LIN {X 0.037,Y -390.880,Z 705.624,A 0.000,B 0.000,C 90.000,E1 148.329} C_DIS
LIN {X -0.098,Y -391.913,Z 705.612,A 0.000,B 0.000,C 90.000,E1 146.215} C_DIS
LIN {X 0.024,Y -394.278,Z 705.595,A 0.000,B 0.000,C 90.000,E1 143.004} C_DIS
LIN {X 0.010,Y -397.554,Z 705.577,A 0.000,B 0.000,C 90.000,E1 139.828} C_DIS
LIN {X -0.151,Y -400.624,Z 705.563,A 0.000,B 0.000,C 90.000,E1 137.391} C_DIS
LIN {X -0.043,Y -401.218,Z 705.561,A 0.000,B 0.000,C 90.000,E1 137.025} C_DIS
LIN {X 0.071,Y -403.273,Z 705.556,A 0.000,B 0.000,C 90.000,E1 136.134} C_DIS
LIN {X -0.018,Y -403.782,Z 705.555,A 0.000,B 0.000,C 90.000,E1 135.972} C_DIS
LIN {X 0.110,Y -405.250,Z 705.553,A 0.000,B 0.000,C 90.000,E1 135.567} C_DIS
LIN {X -0.029,Y -408.274,Z 705.550,A 0.000,B 0.000,C 90.000,E1 135.040} C_DIS
LIN {X -0.096,Y -412.512,Z 705.547,A 0.000,B 0.000,C 90.000,E1 134.514} C_DIS
LIN {X 0.208,Y -421.421,Z 705.542,A 0.000,B 0.000,C 90.000,E1 133.542} C_DIS
LIN {X -0.002,Y -435.121,Z 705.535,A 0.000,B 0.000,C 90.000,E1 132.285} C_DIS
LIN {X 0.155,Y -448.848,Z 705.528,A 0.000,B 0.000,C 90.000,E1 131.067} C_DIS
LIN {X 0.075,Y -459.384,Z 705.523,A 0.000,B 0.000,C 90.000,E1 130.172} C_DIS
LIN {X -0.134,Y -469.829,Z 705.518,A 0.000,B 0.000,C 90.000,E1 129.277} C_DIS
LIN {X 0.058,Y -477.114,Z 705.514,A 0.000,B 0.000,C 90.000,E1 128.588} C_DIS
LIN {X 0.072,Y -486.841,Z 705.509,A 0.000,B 0.000,C 90.000,E1 127.649} C_DIS
LIN {X 0.054,Y -494.993,Z 705.505,A 0.000,B 0.000,C 90.000,E1 126.824} C_DIS
LIN {X -0.059,Y -501.689,Z 705.501,A 0.000,B 0.000,C 90.000,E1 126.137} C_DIS
LIN {X 0.320,Y -506.811,Z 705.498,A 0.000,B 0.000,C 90.000,E1 125.518} C_DIS
LIN {X 0.021,Y -510.602,Z 705.495,A 0.000,B 0.000,C 90.000,E1 125.105} C_DIS
LIN {X -0.156,Y -515.288,Z 705.492,A 0.000,B 0.000,C 90.000,E1 124.532} C_DIS
LIN {X -0.052,Y -520.560,Z 705.488,A 0.000,B 0.000,C 90.000,E1 123.785} C_DIS
LIN {X -0.281,Y -523.579,Z 705.485,A 0.000,B 0.000,C 90.000,E1 123.372} C_DIS
LIN {X -0.096,Y -528.125,Z 705.481,A 0.000,B 0.000,C 90.000,E1 122.625} C_DIS
LIN {X 0.290,Y -531.521,Z 705.478,A 0.000,B 0.000,C 90.000,E1 122.005} C_DIS
LIN {X -0.160,Y -535.306,Z 705.474,A 0.000,B 0.000,C 90.000,E1 121.337} C_DIS
LIN {X 0.156,Y -538.794,Z 705.470,A 0.000,B 0.000,C 90.000,E1 120.590} C_DIS
LIN {X -0.053,Y -543.188,Z 705.465,A 0.000,B 0.000,C 90.000,E1 119.617} C_DIS
LIN {X -0.177,Y -545.069,Z 705.462,A 0.000,B 0.000,C 90.000,E1 119.205} C_DIS
LIN {X 0.052,Y -549.671,Z 705.456,A 0.000,B 0.000,C 90.000,E1 118.052} C_DIS
LIN {X 0.114,Y -553.949,Z 705.450,A 0.000,B 0.000,C 90.000,E1 116.924} C_DIS
LIN {X -0.274,Y -557.841,Z 705.443,A 0.000,B 0.000,C 90.000,E1 115.848} C_DIS
LIN {X 0.106,Y -560.454,Z 705.439,A 0.000,B 0.000,C 90.000,E1 114.975} C_DIS
LIN {X -0.301,Y -562.053,Z 705.436,A 0.000,B 0.000,C 90.000,E1 114.463} C_DIS
LIN {X -0.060,Y -564.908,Z 705.430,A 0.000,B 0.000,C 90.000,E1 113.334} C_DIS
LIN {X -0.116,Y -566.717,Z 705.425,A 0.000,B 0.000,C 90.000,E1 112.514} C_DIS
LIN {X -0.032,Y -568.729,Z 705.419,A 0.000,B 0.000,C 90.000,E1 111.408} C_DIS
LIN {X 0.084,Y -570.665,Z 705.413,A 0.000,B 0.000,C 90.000,E1 110.301} C_DIS
LIN {X -0.170,Y -573.851,Z 705.402,A 0.000,B 0.000,C 90.000,E1 108.417} C_DIS
LIN {X -0.347,Y -576.446,Z 705.393,A 0.000,B 0.000,C 90.000,E1 106.804} C_DIS
LIN {X 0.230,Y -578.049,Z 705.387,A 0.000,B 0.000,C 90.000,E1 105.662} C_DIS
LIN {X -0.232,Y -580.067,Z 705.380,A 0.000,B 0.000,C 90.000,E1 104.356} C_DIS
LIN {X -0.237,Y -582.029,Z 705.372,A 0.000,B 0.000,C 90.000,E1 103.008} C_DIS
LIN {X -0.290,Y -584.774,Z 705.362,A 0.000,B 0.000,C 90.000,E1 101.130} C_DIS
LIN {X -0.218,Y -586.749,Z 705.354,A 0.000,B 0.000,C 90.000,E1 99.782} C_DIS
LIN {X 0.270,Y -588.417,Z 705.347,A 0.000,B 0.000,C 90.000,E1 98.398} C_DIS
LIN {X -0.113,Y -590.377,Z 705.338,A 0.000,B 0.000,C 90.000,E1 96.834} C_DIS
LIN {X 0.052,Y -592.186,Z 705.329,A 0.000,B 0.000,C 90.000,E1 95.220} C_DIS
LIN {X -0.008,Y -593.656,Z 705.322,A 0.000,B 0.000,C 90.000,E1 93.898} C_DIS
LIN {X 0.293,Y -594.679,Z 705.316,A 0.000,B 0.000,C 90.000,E1 92.808} C_DIS
LIN {X 0.237,Y -595.838,Z 705.308,A 0.000,B 0.000,C 90.000,E1 91.489} C_DIS
LIN {X 0.186,Y -596.766,Z 705.301,A 0.000,B 0.000,C 90.000,E1 90.172} C_DIS
LIN {X -0.081,Y -597.292,Z 705.295,A 0.000,B 0.000,C 90.000,E1 89.141} C_DIS
LIN {X 0.142,Y -597.849,Z 705.286,A 0.000,B 0.000,C 90.000,E1 87.535} C_DIS
LIN {X 0.138,Y -598.168,Z 705.279,A 0.000,B 0.000,C 90.000,E1 86.216} C_DIS
LIN {X -0.192,Y -598.390,Z 705.270,A 0.000,B 0.000,C 90.000,E1 84.666} C_DIS
LIN {X 0.221,Y -598.369,Z 705.264,A 0.000,B 0.000,C 90.000,E1 83.571} C_DIS
LIN {X 0.026,Y -598.147,Z 705.256,A 0.000,B 0.000,C 90.000,E1 82.008} C_DIS
LIN {X -0.165,Y -597.774,Z 705.250,A 0.000,B 0.000,C 90.000,E1 80.971} C_DIS
LIN {X -0.274,Y -597.248,Z 705.244,A 0.000,B 0.000,C 90.000,E1 79.926} C_DIS
LIN {X 0.300,Y -596.197,Z 705.235,A 0.000,B 0.000,C 90.000,E1 78.285} C_DIS
LIN {X -0.005,Y -595.130,Z 705.228,A 0.000,B 0.000,C 90.000,E1 76.992} C_DIS
LIN {X -0.033,Y -594.149,Z 705.222,A 0.000,B 0.000,C 90.000,E1 75.936} C_DIS
LIN {X 0.069,Y -593.162,Z 705.216,A 0.000,B 0.000,C 90.000,E1 74.866} C_DIS
LIN {X -0.146,Y -591.785,Z 705.209,A 0.000,B 0.000,C 90.000,E1 73.559} C_DIS
LIN {X 0.030,Y -589.941,Z 705.200,A 0.000,B 0.000,C 90.000,E1 71.945} C_DIS
LIN {X 0.242,Y -588.599,Z 705.194,A 0.000,B 0.000,C 90.000,E1 70.859} C_DIS
LIN {X -0.252,Y -586.709,Z 705.186,A 0.000,B 0.000,C 90.000,E1 69.571} C_DIS
LIN {X 0.117,Y -585.109,Z 705.180,A 0.000,B 0.000,C 90.000,E1 68.465} C_DIS
LIN {X -0.078,Y -583.265,Z 705.174,A 0.000,B 0.000,C 90.000,E1 67.411} C_DIS
LIN {X -0.167,Y -581.732,Z 705.170,A 0.000,B 0.000,C 90.000,E1 66.613} C_DIS
LIN {X -0.178,Y -579.515,Z 705.164,A 0.000,B 0.000,C 90.000,E1 65.537} C_DIS
LIN {X -0.073,Y -577.612,Z 705.160,A 0.000,B 0.000,C 90.000,E1 64.717} C_DIS
LIN {X -0.140,Y -574.784,Z 705.154,A 0.000,B 0.000,C 90.000,E1 63.640} C_DIS
LIN {X 0.009,Y -571.694,Z 705.147,A 0.000,B 0.000,C 90.000,E1 62.538} C_DIS
LIN {X 0.115,Y -568.247,Z 705.141,A 0.000,B 0.000,C 90.000,E1 61.435} C_DIS
LIN {X -0.237,Y -566.465,Z 705.138,A 0.000,B 0.000,C 90.000,E1 60.923} C_DIS
LIN {X -0.021,Y -563.520,Z 705.134,A 0.000,B 0.000,C 90.000,E1 60.078} C_DIS
LIN {X -0.042,Y -560.328,Z 705.129,A 0.000,B 0.000,C 90.000,E1 59.253} C_DIS
LIN {X 0.207,Y -557.352,Z 705.125,A 0.000,B 0.000,C 90.000,E1 58.535} C_DIS
LIN {X -0.055,Y -554.041,Z 705.122,A 0.000,B 0.000,C 90.000,E1 57.867} C_DIS
LIN {X -0.051,Y -550.348,Z 705.118,A 0.000,B 0.000,C 90.000,E1 57.168} C_DIS
LIN {X 0.253,Y -545.320,Z 705.113,A 0.000,B 0.000,C 90.000,E1 56.294} C_DIS
LIN {X 0.155,Y -542.697,Z 705.111,A 0.000,B 0.000,C 90.000,E1 55.881} C_DIS
LIN {X 0.063,Y -537.718,Z 705.107,A 0.000,B 0.000,C 90.000,E1 55.182} C_DIS
LIN {X -0.074,Y -534.597,Z 705.104,A 0.000,B 0.000,C 90.000,E1 54.769} C_DIS
LIN {X -0.076,Y -529.880,Z 705.101,A 0.000,B 0.000,C 90.000,E1 54.196} C_DIS
LIN {X -0.045,Y -524.667,Z 705.098,A 0.000,B 0.000,C 90.000,E1 53.623} C_DIS
LIN {X -0.063,Y -520.475,Z 705.096,A 0.000,B 0.000,C 90.000,E1 53.210} C_DIS
LIN {X -0.293,Y -516.009,Z 705.093,A 0.000,B 0.000,C 90.000,E1 52.844} C_DIS
LIN {X 0.063,Y -509.957,Z 705.091,A 0.000,B 0.000,C 90.000,E1 52.316} C_DIS
LIN {X -0.087,Y -505.088,Z 705.089,A 0.000,B 0.000,C 90.000,E1 51.984} C_DIS
LIN {X 0.054,Y -498.624,Z 705.086,A 0.000,B 0.000,C 90.000,E1 51.537} C_DIS
LIN {X -0.018,Y -490.654,Z 705.084,A 0.000,B 0.000,C 90.000,E1 51.045} C_DIS
LIN {X -0.006,Y -473.974,Z 705.078,A 0.000,B 0.000,C 90.000,E1 50.070} C_DIS
LIN {X 0.267,Y -454.288,Z 705.072,A 0.000,B 0.000,C 90.000,E1 48.852} C_DIS
LIN {X 0.001,Y -431.613,Z 705.064,A 0.000,B 0.000,C 90.000,E1 47.433} C_DIS
LIN {X -0.119,Y -422.494,Z 705.060,A 0.000,B 0.000,C 90.000,E1 46.782} C_DIS
LIN {X -0.020,Y -422.180,Z 705.060,A 0.000,B 0.000,C 90.000,E1 46.743} C_DIS
LIN {X -0.043,Y -422.169,Z 705.060,A 0.000,B 0.000,C 90.000,E1 46.743} C_DIS
LIN {X 0.214,Y -418.724,Z 705.049,A 0.000,B 0.000,C 90.000,E1 44.838} C_DIS
LIN {X -0.192,Y -409.471,Z 705.026,A 0.000,B 0.000,C 90.000,E1 40.620} C_DIS
LIN {X -0.082,Y -409.331,Z 705.024,A 0.000,B 0.000,C 90.000,E1 40.253} C_DIS
LIN {X 0.119,Y -409.487,Z 705.010,A 0.000,B 0.000,C 90.000,E1 37.810} C_DIS
LIN {X -0.114,Y -410.476,Z 704.993,A 0.000,B 0.000,C 90.000,E1 34.739} C_DIS
LIN {X -0.195,Y -411.108,Z 704.985,A 0.000,B 0.000,C 90.000,E1 33.372} C_DIS
LIN {X 0.026,Y -412.489,Z 704.970,A 0.000,B 0.000,C 90.000,E1 30.590} C_DIS
LIN {X 0.021,Y -413.990,Z 704.955,A 0.000,B 0.000,C 90.000,E1 27.847} C_DIS
LIN {X -0.006,Y -416.018,Z 704.938,A 0.000,B 0.000,C 90.000,E1 24.771} C_DIS
LIN {X -0.025,Y -417.955,Z 704.924,A 0.000,B 0.000,C 90.000,E1 22.386} C_DIS
LIN {X 0.140,Y -419.568,Z 704.915,A 0.000,B 0.000,C 90.000,E1 20.663} C_DIS
LIN {X 0.007,Y -421.974,Z 704.902,A 0.000,B 0.000,C 90.000,E1 18.308} C_DIS
LIN {X -0.081,Y -423.524,Z 704.894,A 0.000,B 0.000,C 90.000,E1 16.968} C_DIS
LIN {X 0.053,Y -426.313,Z 704.881,A 0.000,B 0.000,C 90.000,E1 14.592} C_DIS
LIN {X -0.033,Y -428.873,Z 704.870,A 0.000,B 0.000,C 90.000,E1 12.591} C_DIS
LIN {X 0.161,Y -431.052,Z 704.861,A 0.000,B 0.000,C 90.000,E1 10.894} C_DIS
LIN {X 0.139,Y -434.153,Z 704.848,A 0.000,B 0.000,C 90.000,E1 8.568} C_DIS
LIN {X -0.061,Y -436.899,Z 704.837,A 0.000,B 0.000,C 90.000,E1 6.606} C_DIS
LIN {X -0.198,Y -439.673,Z 704.826,A 0.000,B 0.000,C 90.000,E1 4.645} C_DIS
LIN {X -0.168,Y -441.687,Z 704.818,A 0.000,B 0.000,C 90.000,E1 3.326} C_DIS
LIN {X 0.175,Y -444.903,Z 704.807,A 0.000,B 0.000,C 90.000,E1 1.318} C_DIS
LIN {X -0.131,Y -448.220,Z 704.797,A 0.000,B 0.000,C 90.000,E1 359.484} C_DIS
LIN {X 0.198,Y -451.315,Z 704.788,A 0.000,B 0.000,C 90.000,E1 357.822} C_DIS
LIN {X 0.053,Y -455.759,Z 704.776,A 0.000,B 0.000,C 90.000,E1 355.584} C_DIS
LIN {X 0.099,Y -460.321,Z 704.763,A 0.000,B 0.000,C 90.000,E1 353.337} C_DIS
LIN {X -0.184,Y -463.478,Z 704.754,A 0.000,B 0.000,C 90.000,E1 351.781} C_DIS
LIN {X -0.078,Y -465.958,Z 704.747,A 0.000,B 0.000,C 90.000,E1 350.500} C_DIS
LIN {X -0.111,Y -468.963,Z 704.738,A 0.000,B 0.000,C 90.000,E1 348.926} C_DIS
LIN {X 0.083,Y -471.257,Z 704.731,A 0.000,B 0.000,C 90.000,E1 347.645} C_DIS
LIN {X 0.181,Y -474.654,Z 704.721,A 0.000,B 0.000,C 90.000,E1 345.755} C_DIS
LIN {X 0.061,Y -477.553,Z 704.712,A 0.000,B 0.000,C 90.000,E1 344.212} C_DIS
LIN {X -0.015,Y -480.523,Z 704.704,A 0.000,B 0.000,C 90.000,E1 342.670} C_DIS
LIN {X 0.098,Y -484.927,Z 704.692,A 0.000,B 0.000,C 90.000,E1 340.496} C_DIS
LIN {X 0.056,Y -490.130,Z 704.678,A 0.000,B 0.000,C 90.000,E1 338.050} C_DIS
LIN {X 0.114,Y -491.805,Z 704.675,A 0.000,B 0.000,C 90.000,E1 337.433} C_DIS
LIN {X 0.130,Y -493.357,Z 704.672,A 0.000,B 0.000,C 90.000,E1 336.975} C_DIS
LIN {X 0.172,Y -494.686,Z 704.671,A 0.000,B 0.000,C 90.000,E1 336.666} C_DIS
LIN {X 0.218,Y -496.414,Z 704.669,A 0.000,B 0.000,C 90.000,E1 336.357} C_DIS
LIN {X -0.136,Y -500.322,Z 704.666,A 0.000,B 0.000,C 90.000,E1 335.921} C_DIS
LIN {X 0.058,Y -507.384,Z 704.663,A 0.000,B 0.000,C 90.000,E1 335.281} C_DIS
LIN {X -0.130,Y -514.500,Z 704.660,A 0.000,B 0.000,C 90.000,E1 334.793} C_DIS
LIN {X -0.057,Y -527.150,Z 704.655,A 0.000,B 0.000,C 90.000,E1 333.948} C_DIS
LIN {X 0.013,Y -537.986,Z 704.651,A 0.000,B 0.000,C 90.000,E1 333.204} C_DIS
LIN {X 0.154,Y -543.938,Z 704.649,A 0.000,B 0.000,C 90.000,E1 332.743} C_DIS
LIN {X 0.171,Y -549.794,Z 704.646,A 0.000,B 0.000,C 90.000,E1 332.281} C_DIS
LIN {X -0.049,Y -555.364,Z 704.643,A 0.000,B 0.000,C 90.000,E1 331.820} C_DIS
LIN {X 0.078,Y -559.491,Z 704.641,A 0.000,B 0.000,C 90.000,E1 331.435} C_DIS
LIN {X 0.122,Y -566.010,Z 704.638,A 0.000,B 0.000,C 90.000,E1 330.795} C_DIS
LIN {X 0.253,Y -572.386,Z 704.634,A 0.000,B 0.000,C 90.000,E1 330.127} C_DIS
LIN {X -0.018,Y -578.608,Z 704.631,A 0.000,B 0.000,C 90.000,E1 329.488} C_DIS
LIN {X 0.281,Y -585.780,Z 704.626,A 0.000,B 0.000,C 90.000,E1 328.663} C_DIS
LIN {X -0.239,Y -595.015,Z 704.620,A 0.000,B 0.000,C 90.000,E1 327.661} C_DIS
LIN {X 0.105,Y -601.689,Z 704.616,A 0.000,B 0.000,C 90.000,E1 326.834} C_DIS
LIN {X -0.133,Y -605.781,Z 704.613,A 0.000,B 0.000,C 90.000,E1 326.342} C_DIS
LIN {X -0.014,Y -611.762,Z 704.609,A 0.000,B 0.000,C 90.000,E1 325.548} C_DIS
LIN {X 0.032,Y -616.458,Z 704.605,A 0.000,B 0.000,C 90.000,E1 324.895} C_DIS
LIN {X 0.083,Y -622.649,Z 704.600,A 0.000,B 0.000,C 90.000,E1 323.989} C_DIS
LIN {X 0.216,Y -627.607,Z 704.596,A 0.000,B 0.000,C 90.000,E1 323.210} C_DIS
LIN {X -0.113,Y -632.970,Z 704.591,A 0.000,B 0.000,C 90.000,E1 322.351} C_DIS
LIN {X 0.003,Y -638.866,Z 704.585,A 0.000,B 0.000,C 90.000,E1 321.331} C_DIS
LIN {X -0.301,Y -644.423,Z 704.580,A 0.000,B 0.000,C 90.000,E1 320.356} C_DIS
LIN {X -0.039,Y -649.734,Z 704.574,A 0.000,B 0.000,C 90.000,E1 319.337} C_DIS
LIN {X 0.182,Y -655.946,Z 704.567,A 0.000,B 0.000,C 90.000,E1 318.081} C_DIS
LIN {X 0.082,Y -660.015,Z 704.563,A 0.000,B 0.000,C 90.000,E1 317.229} C_DIS
LIN {X 0.019,Y -663.227,Z 704.558,A 0.000,B 0.000,C 90.000,E1 316.500} C_DIS
LIN {X 0.000,Y -667.217,Z 704.553,A 0.000,B 0.000,C 90.000,E1 315.526} C_DIS
LIN {X 0.021,Y -671.839,Z 704.546,A 0.000,B 0.000,C 90.000,E1 314.312} C_DIS
LIN {X 0.115,Y -675.298,Z 704.541,A 0.000,B 0.000,C 90.000,E1 313.338} C_DIS
LIN {X -0.191,Y -679.496,Z 704.534,A 0.000,B 0.000,C 90.000,E1 312.162} C_DIS
LIN {X -0.035,Y -682.652,Z 704.529,A 0.000,B 0.000,C 90.000,E1 311.191} C_DIS
LIN {X -0.225,Y -685.529,Z 704.524,A 0.000,B 0.000,C 90.000,E1 310.253} C_DIS
LIN {X -0.125,Y -686.898,Z 704.521,A 0.000,B 0.000,C 90.000,E1 309.769} C_DIS
LIN {X -0.252,Y -689.277,Z 704.516,A 0.000,B 0.000,C 90.000,E1 308.830} C_DIS
LIN {X -0.030,Y -690.417,Z 704.513,A 0.000,B 0.000,C 90.000,E1 308.338} C_DIS
LIN {X -0.041,Y -692.780,Z 704.506,A 0.000,B 0.000,C 90.000,E1 307.156} C_DIS
LIN {X 0.119,Y -694.865,Z 704.500,A 0.000,B 0.000,C 90.000,E1 305.964} C_DIS
LIN {X 0.095,Y -696.266,Z 704.495,A 0.000,B 0.000,C 90.000,E1 305.025} C_DIS
LIN {X -0.083,Y -697.758,Z 704.488,A 0.000,B 0.000,C 90.000,E1 303.865} C_DIS
LIN {X -0.137,Y -698.550,Z 704.484,A 0.000,B 0.000,C 90.000,E1 303.166} C_DIS
LIN {X -0.279,Y -699.602,Z 704.478,A 0.000,B 0.000,C 90.000,E1 302.005} C_DIS
LIN {X -0.073,Y -700.436,Z 704.473,A 0.000,B 0.000,C 90.000,E1 301.052} C_DIS
LIN {X -0.220,Y -701.001,Z 704.467,A 0.000,B 0.000,C 90.000,E1 300.129} C_DIS
LIN {X 0.188,Y -701.519,Z 704.460,A 0.000,B 0.000,C 90.000,E1 298.693} C_DIS
LIN {X -0.014,Y -702.026,Z 704.452,A 0.000,B 0.000,C 90.000,E1 297.308} C_DIS
LIN {X 0.057,Y -702.907,Z 704.443,A 0.000,B 0.000,C 90.000,E1 295.668} C_DIS
LIN {X -0.016,Y -702.981,Z 704.440,A 0.000,B 0.000,C 90.000,E1 295.207} C_DIS
LIN {X 0.264,Y -702.814,Z 704.439,A 0.000,B 0.000,C 90.000,E1 294.951} C_DIS
LIN {X -0.110,Y -702.105,Z 704.436,A 0.000,B 0.000,C 90.000,E1 294.515} C_DIS
LIN {X 0.167,Y -701.179,Z 704.435,A 0.000,B 0.000,C 90.000,E1 294.259} C_DIS
LIN {X 0.156,Y -699.848,Z 704.434,A 0.000,B 0.000,C 90.000,E1 294.027} C_DIS
LIN {X -0.214,Y -698.290,Z 704.432,A 0.000,B 0.000,C 90.000,E1 293.823} C_DIS
LIN {X -0.083,Y -697.321,Z 704.432,A 0.000,B 0.000,C 90.000,E1 293.695} C_DIS
LIN {X 0.049,Y -695.872,Z 704.431,A 0.000,B 0.000,C 90.000,E1 293.567} C_DIS
LIN {X 0.294,Y -692.126,Z 704.430,A 0.000,B 0.000,C 90.000,E1 293.334} C_DIS
LIN {X -0.230,Y -688.625,Z 704.429,A 0.000,B 0.000,C 90.000,E1 293.206} C_DIS
LIN {X -0.232,Y -686.655,Z 704.428,A 0.000,B 0.000,C 90.000,E1 293.131} C_DIS
LIN {X 0.049,Y -679.403,Z 704.428,A 0.000,B 0.000,C 90.000,E1 292.950} C_DIS
LIN {X 0.238,Y -677.497,Z 704.427,A 0.000,B 0.000,C 90.000,E1 292.898} C_DIS
LIN {X -0.265,Y -663.430,Z 704.426,A 0.000,B 0.000,C 90.000,E1 292.770} C_DIS
LIN {X 0.219,Y -646.156,Z 704.425,A 0.000,B 0.000,C 90.000,E1 292.461} C_DIS
LIN {X 0.166,Y -636.385,Z 704.424,A 0.000,B 0.000,C 90.000,E1 292.280} C_DIS
LIN {X -0.090,Y -626.375,Z 704.423,A 0.000,B 0.000,C 90.000,E1 292.078} C_DIS
LIN {X -0.162,Y -609.548,Z 704.420,A 0.000,B 0.000,C 90.000,E1 291.642} C_DIS
LIN {X -0.164,Y -574.898,Z 704.414,A 0.000,B 0.000,C 90.000,E1 290.610} C_DIS
LIN {X 0.112,Y -567.673,Z 704.413,A 0.000,B 0.000,C 90.000,E1 290.375} C_DIS
LIN {X 0.009,Y -560.839,Z 704.412,A 0.000,B 0.000,C 90.000,E1 290.120} C_DIS
LIN {X -0.104,Y -559.411,Z 704.411,A 0.000,B 0.000,C 90.000,E1 290.066} C_DIS
LIN {X 0.165,Y -557.065,Z 704.411,A 0.000,B 0.000,C 90.000,E1 289.885} C_DIS
LIN {X 0.082,Y -556.069,Z 704.410,A 0.000,B 0.000,C 90.000,E1 289.812} C_DIS
LIN {X 0.041,Y -556.051,Z 704.410,A 0.000,B 0.000,C 90.000,E1 289.812} C_DIS
LIN {X -0.053,Y -555.240,Z 704.409,A 0.000,B 0.000,C 90.000,E1 289.631} C_DIS
LIN {X -0.069,Y -554.659,Z 704.407,A 0.000,B 0.000,C 90.000,E1 289.214} C_DIS
LIN {X 0.214,Y -553.944,Z 704.397,A 0.000,B 0.000,C 90.000,E1 287.511} C_DIS
LIN {X 0.144,Y -553.312,Z 704.388,A 0.000,B 0.000,C 90.000,E1 285.843} C_DIS
LIN {X 0.176,Y -552.632,Z 704.377,A 0.000,B 0.000,C 90.000,E1 283.883} C_DIS
LIN {X -0.188,Y -551.995,Z 704.368,A 0.000,B 0.000,C 90.000,E1 282.243} C_DIS
LIN {X -0.021,Y -551.249,Z 704.359,A 0.000,B 0.000,C 90.000,E1 280.546} C_DIS
LIN {X 0.243,Y -550.246,Z 704.346,A 0.000,B 0.000,C 90.000,E1 278.276} C_DIS
LIN {X 0.210,Y -549.520,Z 704.335,A 0.000,B 0.000,C 90.000,E1 276.315} C_DIS
LIN {X 0.111,Y -549.126,Z 704.324,A 0.000,B 0.000,C 90.000,E1 274.359} C_DIS
LIN {X -0.132,Y -548.868,Z 704.317,A 0.000,B 0.000,C 90.000,E1 272.980} C_DIS
LIN {X 0.180,Y -548.340,Z 704.307,A 0.000,B 0.000,C 90.000,E1 271.260} C_DIS
LIN {X -0.220,Y -547.976,Z 704.302,A 0.000,B 0.000,C 90.000,E1 270.458} C_DIS
LIN {X 0.064,Y -546.926,Z 704.293,A 0.000,B 0.000,C 90.000,E1 268.740} C_DIS
LIN {X -0.213,Y -545.935,Z 704.284,A 0.000,B 0.000,C 90.000,E1 267.078} C_DIS
LIN {X 0.060,Y -544.775,Z 704.274,A 0.000,B 0.000,C 90.000,E1 265.355} C_DIS
LIN {X -0.111,Y -543.313,Z 704.263,A 0.000,B 0.000,C 90.000,E1 263.394} C_DIS
LIN {X 0.143,Y -542.023,Z 704.255,A 0.000,B 0.000,C 90.000,E1 261.951} C_DIS
LIN {X -0.028,Y -540.178,Z 704.244,A 0.000,B 0.000,C 90.000,E1 259.982} C_DIS
LIN {X -0.125,Y -538.572,Z 704.235,A 0.000,B 0.000,C 90.000,E1 258.285} C_DIS
LIN {X 0.205,Y -537.294,Z 704.227,A 0.000,B 0.000,C 90.000,E1 256.825} C_DIS
LIN {X 0.156,Y -535.749,Z 704.217,A 0.000,B 0.000,C 90.000,E1 255.117} C_DIS
LIN {X -0.071,Y -534.918,Z 704.213,A 0.000,B 0.000,C 90.000,E1 254.283} C_DIS
LIN {X 0.080,Y -533.430,Z 704.205,A 0.000,B 0.000,C 90.000,E1 252.834} C_DIS
LIN {X 0.243,Y -531.726,Z 704.195,A 0.000,B 0.000,C 90.000,E1 251.094} C_DIS
LIN {X 0.140,Y -530.799,Z 704.190,A 0.000,B 0.000,C 90.000,E1 250.242} C_DIS
LIN {X -0.101,Y -528.521,Z 704.181,A 0.000,B 0.000,C 90.000,E1 248.539} C_DIS
LIN {X 0.130,Y -526.859,Z 704.174,A 0.000,B 0.000,C 90.000,E1 247.358} C_DIS
LIN {X -0.145,Y -525.206,Z 704.168,A 0.000,B 0.000,C 90.000,E1 246.230} C_DIS
LIN {X 0.097,Y -522.309,Z 704.158,A 0.000,B 0.000,C 90.000,E1 244.460} C_DIS
LIN {X 0.075,Y -520.780,Z 704.153,A 0.000,B 0.000,C 90.000,E1 243.589} C_DIS
LIN {X -0.157,Y -518.027,Z 704.145,A 0.000,B 0.000,C 90.000,E1 242.153} C_DIS
LIN {X 0.020,Y -515.150,Z 704.137,A 0.000,B 0.000,C 90.000,E1 240.667} C_DIS
LIN {X -0.057,Y -512.044,Z 704.129,A 0.000,B 0.000,C 90.000,E1 239.203} C_DIS
LIN {X -0.290,Y -508.285,Z 704.119,A 0.000,B 0.000,C 90.000,E1 237.454} C_DIS
LIN {X -0.049,Y -504.422,Z 704.109,A 0.000,B 0.000,C 90.000,E1 235.642} C_DIS
LIN {X 0.224,Y -501.153,Z 704.101,A 0.000,B 0.000,C 90.000,E1 234.116} C_DIS
LIN {X -0.130,Y -498.946,Z 704.096,A 0.000,B 0.000,C 90.000,E1 233.256} C_DIS
LIN {X -0.213,Y -494.272,Z 704.086,A 0.000,B 0.000,C 90.000,E1 231.457} C_DIS
LIN {X 0.057,Y -489.099,Z 704.074,A 0.000,B 0.000,C 90.000,E1 229.299} C_DIS
LIN {X 0.026,Y -486.242,Z 704.067,A 0.000,B 0.000,C 90.000,E1 228.081} C_DIS
LIN {X 0.221,Y -482.083,Z 704.057,A 0.000,B 0.000,C 90.000,E1 226.215} C_DIS
LIN {X -0.253,Y -477.289,Z 704.045,A 0.000,B 0.000,C 90.000,E1 224.109} C_DIS
LIN {X 0.015,Y -471.128,Z 704.029,A 0.000,B 0.000,C 90.000,E1 221.272} C_DIS
LIN {X 0.030,Y -466.427,Z 704.017,A 0.000,B 0.000,C 90.000,E1 219.072} C_DIS
LIN {X 0.019,Y -463.688,Z 704.010,A 0.000,B 0.000,C 90.000,E1 217.810} C_DIS
LIN {X 0.070,Y -460.299,Z 704.001,A 0.000,B 0.000,C 90.000,E1 216.217} C_DIS
LIN {X 0.099,Y -455.361,Z 703.987,A 0.000,B 0.000,C 90.000,E1 213.658} C_DIS
LIN {X -0.062,Y -451.660,Z 703.976,A 0.000,B 0.000,C 90.000,E1 211.750} C_DIS
LIN {X 0.139,Y -447.438,Z 703.964,A 0.000,B 0.000,C 90.000,E1 209.461} C_DIS
LIN {X 0.105,Y -443.941,Z 703.953,A 0.000,B 0.000,C 90.000,E1 207.513} C_DIS
LIN {X -0.210,Y -440.326,Z 703.942,A 0.000,B 0.000,C 90.000,E1 205.591} C_DIS
LIN {X 0.166,Y -437.338,Z 703.933,A 0.000,B 0.000,C 90.000,E1 203.898} C_DIS
LIN {X -0.088,Y -434.309,Z 703.924,A 0.000,B 0.000,C 90.000,E1 202.280} C_DIS
LIN {X -0.002,Y -431.301,Z 703.915,A 0.000,B 0.000,C 90.000,E1 200.610} C_DIS
LIN {X 0.073,Y -427.704,Z 703.903,A 0.000,B 0.000,C 90.000,E1 198.598} C_DIS
LIN {X -0.017,Y -423.406,Z 703.890,A 0.000,B 0.000,C 90.000,E1 196.260} C_DIS
LIN {X -0.103,Y -419.694,Z 703.879,A 0.000,B 0.000,C 90.000,E1 194.245} C_DIS
LIN {X 0.036,Y -416.149,Z 703.868,A 0.000,B 0.000,C 90.000,E1 192.187} C_DIS
LIN {X 0.002,Y -412.660,Z 703.856,A 0.000,B 0.000,C 90.000,E1 190.141} C_DIS
LIN {X -0.143,Y -408.246,Z 703.841,A 0.000,B 0.000,C 90.000,E1 187.409} C_DIS
LIN {X -0.156,Y -405.185,Z 703.830,A 0.000,B 0.000,C 90.000,E1 185.334} C_DIS
LIN {X 0.077,Y -401.741,Z 703.816,A 0.000,B 0.000,C 90.000,E1 182.865} C_DIS
LIN {X 0.130,Y -398.448,Z 703.800,A 0.000,B 0.000,C 90.000,E1 180.057} C_DIS
LIN {X -0.030,Y -395.063,Z 703.781,A 0.000,B 0.000,C 90.000,E1 176.560} C_DIS
LIN {X 0.009,Y -392.171,Z 703.755,A 0.000,B 0.000,C 90.000,E1 171.951} C_DIS
LIN {X 0.173,Y -391.450,Z 703.745,A 0.000,B 0.000,C 90.000,E1 170.151} C_DIS
LIN {X -0.093,Y -390.705,Z 703.732,A 0.000,B 0.000,C 90.000,E1 167.701} C_DIS
LIN {X 0.222,Y -390.083,Z 703.720,A 0.000,B 0.000,C 90.000,E1 165.519} C_DIS
LIN {X -0.168,Y -389.756,Z 703.710,A 0.000,B 0.000,C 90.000,E1 163.795} C_DIS
LIN {X -0.005,Y -389.538,Z 703.696,A 0.000,B 0.000,C 90.000,E1 161.275} C_DIS
LIN {X -0.004,Y -389.511,Z 703.684,A 0.000,B 0.000,C 90.000,E1 159.135} C_DIS
LIN {X -0.158,Y -389.657,Z 703.668,A 0.000,B 0.000,C 90.000,E1 156.305} C_DIS
LIN {X 0.125,Y -389.951,Z 703.654,A 0.000,B 0.000,C 90.000,E1 153.768} C_DIS
LIN {X -0.141,Y -390.193,Z 703.645,A 0.000,B 0.000,C 90.000,E1 152.025} C_DIS
LIN {X -0.085,Y -391.115,Z 703.625,A 0.000,B 0.000,C 90.000,E1 148.456} C_DIS
LIN {X 0.048,Y -393.245,Z 703.603,A 0.000,B 0.000,C 90.000,E1 144.529} C_DIS
LIN {X 0.136,Y -395.989,Z 703.585,A 0.000,B 0.000,C 90.000,E1 141.331} C_DIS
LIN {X 0.125,Y -398.231,Z 703.574,A 0.000,B 0.000,C 90.000,E1 139.218} C_DIS
LIN {X -0.127,Y -400.920,Z 703.562,A 0.000,B 0.000,C 90.000,E1 137.148} C_DIS
LIN {X -0.018,Y -401.552,Z 703.560,A 0.000,B 0.000,C 90.000,E1 136.782} C_DIS
LIN {X -0.098,Y -402.372,Z 703.558,A 0.000,B 0.000,C 90.000,E1 136.458} C_DIS
LIN {X 0.002,Y -403.070,Z 703.556,A 0.000,B 0.000,C 90.000,E1 136.095} C_DIS
LIN {X -0.053,Y -405.410,Z 703.552,A 0.000,B 0.000,C 90.000,E1 135.405} C_DIS
LIN {X -0.016,Y -408.244,Z 703.549,A 0.000,B 0.000,C 90.000,E1 134.879} C_DIS
LIN {X 0.052,Y -412.342,Z 703.547,A 0.000,B 0.000,C 90.000,E1 134.352} C_DIS
LIN {X 0.050,Y -420.408,Z 703.542,A 0.000,B 0.000,C 90.000,E1 133.500} C_DIS
LIN {X -0.053,Y -432.583,Z 703.535,A 0.000,B 0.000,C 90.000,E1 132.366} C_DIS
LIN {X -0.077,Y -449.392,Z 703.527,A 0.000,B 0.000,C 90.000,E1 130.906} C_DIS
LIN {X 0.201,Y -458.537,Z 703.523,A 0.000,B 0.000,C 90.000,E1 130.092} C_DIS
LIN {X -0.039,Y -470.502,Z 703.517,A 0.000,B 0.000,C 90.000,E1 129.072} C_DIS
LIN {X 0.181,Y -477.744,Z 703.513,A 0.000,B 0.000,C 90.000,E1 128.382} C_DIS
LIN {X -0.172,Y -486.334,Z 703.509,A 0.000,B 0.000,C 90.000,E1 127.604} C_DIS
LIN {X 0.215,Y -493.213,Z 703.505,A 0.000,B 0.000,C 90.000,E1 126.870} C_DIS
LIN {X 0.169,Y -500.048,Z 703.501,A 0.000,B 0.000,C 90.000,E1 126.171} C_DIS
LIN {X 0.109,Y -506.458,Z 703.497,A 0.000,B 0.000,C 90.000,E1 125.471} C_DIS
LIN {X 0.049,Y -511.339,Z 703.494,A 0.000,B 0.000,C 90.000,E1 124.898} C_DIS
LIN {X 0.065,Y -514.907,Z 703.492,A 0.000,B 0.000,C 90.000,E1 124.452} C_DIS
LIN {X 0.055,Y -519.281,Z 703.488,A 0.000,B 0.000,C 90.000,E1 123.865} C_DIS
LIN {X -0.065,Y -523.373,Z 703.485,A 0.000,B 0.000,C 90.000,E1 123.293} C_DIS
LIN {X -0.003,Y -527.134,Z 703.482,A 0.000,B 0.000,C 90.000,E1 122.704} C_DIS
LIN {X -0.228,Y -531.467,Z 703.478,A 0.000,B 0.000,C 90.000,E1 122.005} C_DIS
LIN {X 0.031,Y -535.348,Z 703.474,A 0.000,B 0.000,C 90.000,E1 121.258} C_DIS
LIN {X 0.053,Y -538.886,Z 703.470,A 0.000,B 0.000,C 90.000,E1 120.541} C_DIS
LIN {X 0.248,Y -542.726,Z 703.465,A 0.000,B 0.000,C 90.000,E1 119.667} C_DIS
LIN {X -0.136,Y -545.801,Z 703.461,A 0.000,B 0.000,C 90.000,E1 118.999} C_DIS
LIN {X -0.142,Y -549.325,Z 703.456,A 0.000,B 0.000,C 90.000,E1 118.153} C_DIS
LIN {X -0.114,Y -552.605,Z 703.452,A 0.000,B 0.000,C 90.000,E1 117.308} C_DIS
LIN {X -0.304,Y -555.665,Z 703.447,A 0.000,B 0.000,C 90.000,E1 116.488} C_DIS
LIN {X 0.291,Y -558.565,Z 703.442,A 0.000,B 0.000,C 90.000,E1 115.591} C_DIS
LIN {X 0.173,Y -561.147,Z 703.438,A 0.000,B 0.000,C 90.000,E1 114.771} C_DIS
LIN {X -0.116,Y -564.143,Z 703.432,A 0.000,B 0.000,C 90.000,E1 113.695} C_DIS
LIN {X 0.011,Y -565.533,Z 703.429,A 0.000,B 0.000,C 90.000,E1 113.131} C_DIS
LIN {X -0.260,Y -567.288,Z 703.424,A 0.000,B 0.000,C 90.000,E1 112.333} C_DIS
LIN {X 0.179,Y -569.791,Z 703.416,A 0.000,B 0.000,C 90.000,E1 110.918} C_DIS
LIN {X -0.068,Y -572.160,Z 703.409,A 0.000,B 0.000,C 90.000,E1 109.577} C_DIS
LIN {X 0.264,Y -574.465,Z 703.401,A 0.000,B 0.000,C 90.000,E1 108.181} C_DIS
LIN {X 0.107,Y -577.080,Z 703.392,A 0.000,B 0.000,C 90.000,E1 106.567} C_DIS
LIN {X -0.209,Y -579.076,Z 703.385,A 0.000,B 0.000,C 90.000,E1 105.245} C_DIS
LIN {X 0.131,Y -581.521,Z 703.376,A 0.000,B 0.000,C 90.000,E1 103.592} C_DIS
LIN {X 0.157,Y -583.488,Z 703.368,A 0.000,B 0.000,C 90.000,E1 102.243} C_DIS
LIN {X 0.133,Y -586.286,Z 703.358,A 0.000,B 0.000,C 90.000,E1 100.366} C_DIS
LIN {X -0.127,Y -587.784,Z 703.352,A 0.000,B 0.000,C 90.000,E1 99.321} C_DIS
LIN {X -0.197,Y -589.462,Z 703.344,A 0.000,B 0.000,C 90.000,E1 97.992} C_DIS
LIN {X -0.233,Y -591.091,Z 703.337,A 0.000,B 0.000,C 90.000,E1 96.663} C_DIS
LIN {X -0.048,Y -592.950,Z 703.328,A 0.000,B 0.000,C 90.000,E1 95.049} C_DIS
LIN {X -0.092,Y -594.411,Z 703.321,A 0.000,B 0.000,C 90.000,E1 93.726} C_DIS
LIN {X 0.222,Y -595.398,Z 703.315,A 0.000,B 0.000,C 90.000,E1 92.636} C_DIS
LIN {X 0.178,Y -596.591,Z 703.307,A 0.000,B 0.000,C 90.000,E1 91.318} C_DIS
LIN {X 0.141,Y -597.458,Z 703.300,A 0.000,B 0.000,C 90.000,E1 90.000} C_DIS
LIN {X -0.116,Y -597.962,Z 703.294,A 0.000,B 0.000,C 90.000,E1 88.969} C_DIS
LIN {X 0.118,Y -598.485,Z 703.285,A 0.000,B 0.000,C 90.000,E1 87.364} C_DIS
LIN {X 0.123,Y -598.785,Z 703.278,A 0.000,B 0.000,C 90.000,E1 86.045} C_DIS
LIN {X -0.143,Y -598.961,Z 703.269,A 0.000,B 0.000,C 90.000,E1 84.489} C_DIS
LIN {X -0.088,Y -598.882,Z 703.262,A 0.000,B 0.000,C 90.000,E1 83.166} C_DIS
LIN {X 0.028,Y -598.664,Z 703.255,A 0.000,B 0.000,C 90.000,E1 81.837} C_DIS
LIN {X 0.230,Y -598.097,Z 703.247,A 0.000,B 0.000,C 90.000,E1 80.500} C_DIS
LIN {X -0.165,Y -597.644,Z 703.243,A 0.000,B 0.000,C 90.000,E1 79.746} C_DIS
LIN {X -0.280,Y -596.541,Z 703.234,A 0.000,B 0.000,C 90.000,E1 78.173} C_DIS
LIN {X -0.005,Y -595.419,Z 703.227,A 0.000,B 0.000,C 90.000,E1 76.825} C_DIS
LIN {X -0.173,Y -594.657,Z 703.222,A 0.000,B 0.000,C 90.000,E1 76.047} C_DIS
LIN {X -0.211,Y -593.681,Z 703.217,A 0.000,B 0.000,C 90.000,E1 74.991} C_DIS
LIN {X 0.145,Y -592.251,Z 703.209,A 0.000,B 0.000,C 90.000,E1 73.630} C_DIS
LIN {X -0.061,Y -590.333,Z 703.200,A 0.000,B 0.000,C 90.000,E1 72.054} C_DIS
LIN {X 0.164,Y -589.019,Z 703.194,A 0.000,B 0.000,C 90.000,E1 70.967} C_DIS
LIN {X -0.187,Y -587.485,Z 703.188,A 0.000,B 0.000,C 90.000,E1 69.934} C_DIS
LIN {X -0.145,Y -585.484,Z 703.181,A 0.000,B 0.000,C 90.000,E1 68.592} C_DIS
LIN {X 0.202,Y -583.614,Z 703.175,A 0.000,B 0.000,C 90.000,E1 67.486} C_DIS
LIN {X -0.061,Y -582.625,Z 703.172,A 0.000,B 0.000,C 90.000,E1 66.975} C_DIS
LIN {X 0.098,Y -579.826,Z 703.165,A 0.000,B 0.000,C 90.000,E1 65.613} C_DIS
LIN {X 0.201,Y -577.899,Z 703.160,A 0.000,B 0.000,C 90.000,E1 64.793} C_DIS
LIN {X 0.132,Y -575.013,Z 703.154,A 0.000,B 0.000,C 90.000,E1 63.717} C_DIS
LIN {X -0.073,Y -572.706,Z 703.150,A 0.000,B 0.000,C 90.000,E1 62.922} C_DIS
LIN {X -0.050,Y -570.204,Z 703.145,A 0.000,B 0.000,C 90.000,E1 62.103} C_DIS
LIN {X 0.028,Y -566.619,Z 703.139,A 0.000,B 0.000,C 90.000,E1 61.001} C_DIS
LIN {X -0.249,Y -563.651,Z 703.134,A 0.000,B 0.000,C 90.000,E1 60.205} C_DIS
LIN {X 0.216,Y -560.457,Z 703.130,A 0.000,B 0.000,C 90.000,E1 59.331} C_DIS
LIN {X -0.123,Y -556.764,Z 703.125,A 0.000,B 0.000,C 90.000,E1 58.535} C_DIS
LIN {X -0.095,Y -553.351,Z 703.121,A 0.000,B 0.000,C 90.000,E1 57.837} C_DIS
LIN {X 0.075,Y -549.536,Z 703.117,A 0.000,B 0.000,C 90.000,E1 57.120} C_DIS
LIN {X -0.129,Y -546.211,Z 703.114,A 0.000,B 0.000,C 90.000,E1 56.580} C_DIS
LIN {X 0.021,Y -541.788,Z 703.111,A 0.000,B 0.000,C 90.000,E1 55.881} C_DIS
LIN {X 0.069,Y -537.773,Z 703.107,A 0.000,B 0.000,C 90.000,E1 55.308} C_DIS
LIN {X 0.163,Y -533.787,Z 703.104,A 0.000,B 0.000,C 90.000,E1 54.769} C_DIS
LIN {X 0.175,Y -528.912,Z 703.101,A 0.000,B 0.000,C 90.000,E1 54.196} C_DIS
LIN {X -0.058,Y -524.076,Z 703.098,A 0.000,B 0.000,C 90.000,E1 53.703} C_DIS
LIN {X -0.120,Y -520.199,Z 703.096,A 0.000,B 0.000,C 90.000,E1 53.336} C_DIS
LIN {X -0.284,Y -514.234,Z 703.093,A 0.000,B 0.000,C 90.000,E1 52.844} C_DIS
LIN {X 0.129,Y -509.579,Z 703.091,A 0.000,B 0.000,C 90.000,E1 52.431} C_DIS
LIN {X 0.098,Y -503.081,Z 703.089,A 0.000,B 0.000,C 90.000,E1 51.984} C_DIS
LIN {X 0.123,Y -494.900,Z 703.086,A 0.000,B 0.000,C 90.000,E1 51.457} C_DIS
LIN {X -0.018,Y -489.906,Z 703.084,A 0.000,B 0.000,C 90.000,E1 51.170} C_DIS
LIN {X 0.075,Y -473.373,Z 703.079,A 0.000,B 0.000,C 90.000,E1 50.194} C_DIS
LIN {X 0.173,Y -455.221,Z 703.073,A 0.000,B 0.000,C 90.000,E1 49.094} C_DIS
LIN {X 0.116,Y -434.038,Z 703.065,A 0.000,B 0.000,C 90.000,E1 47.757} C_DIS
LIN {X 0.192,Y -424.462,Z 703.062,A 0.000,B 0.000,C 90.000,E1 47.067} C_DIS
LIN {X -0.024,Y -422.580,Z 703.061,A 0.000,B 0.000,C 90.000,E1 46.944} C_DIS
LIN {X -0.048,Y -422.570,Z 703.061,A 0.000,B 0.000,C 90.000,E1 46.944} C_DIS
LIN {X -0.144,Y -418.448,Z 703.049,A 0.000,B 0.000,C 90.000,E1 44.757} C_DIS
LIN {X 0.172,Y -409.870,Z 703.027,A 0.000,B 0.000,C 90.000,E1 40.782} C_DIS
LIN {X -0.029,Y -409.721,Z 703.025,A 0.000,B 0.000,C 90.000,E1 40.458} C_DIS
LIN {X 0.020,Y -409.824,Z 703.013,A 0.000,B 0.000,C 90.000,E1 38.382} C_DIS
LIN {X -0.045,Y -410.832,Z 702.994,A 0.000,B 0.000,C 90.000,E1 34.945} C_DIS
LIN {X -0.121,Y -411.496,Z 702.987,A 0.000,B 0.000,C 90.000,E1 33.579} C_DIS
LIN {X 0.115,Y -412.840,Z 702.971,A 0.000,B 0.000,C 90.000,E1 30.797} C_DIS
LIN {X 0.021,Y -414.120,Z 702.958,A 0.000,B 0.000,C 90.000,E1 28.409} C_DIS
LIN {X -0.064,Y -414.932,Z 702.950,A 0.000,B 0.000,C 90.000,E1 27.052} C_DIS
LIN {X -0.183,Y -416.858,Z 702.935,A 0.000,B 0.000,C 90.000,E1 24.335} C_DIS
LIN {X -0.107,Y -418.533,Z 702.924,A 0.000,B 0.000,C 90.000,E1 22.280} C_DIS
LIN {X 0.079,Y -420.147,Z 702.914,A 0.000,B 0.000,C 90.000,E1 20.556} C_DIS
LIN {X -0.072,Y -422.198,Z 702.903,A 0.000,B 0.000,C 90.000,E1 18.544} C_DIS
LIN {X -0.100,Y -424.083,Z 702.894,A 0.000,B 0.000,C 90.000,E1 16.858} C_DIS
LIN {X -0.023,Y -426.449,Z 702.882,A 0.000,B 0.000,C 90.000,E1 14.828} C_DIS
LIN {X -0.107,Y -428.952,Z 702.871,A 0.000,B 0.000,C 90.000,E1 12.827} C_DIS
LIN {X 0.090,Y -431.116,Z 702.862,A 0.000,B 0.000,C 90.000,E1 11.130} C_DIS
LIN {X -0.050,Y -433.713,Z 702.851,A 0.000,B 0.000,C 90.000,E1 9.151} C_DIS
LIN {X 0.027,Y -435.440,Z 702.844,A 0.000,B 0.000,C 90.000,E1 7.814} C_DIS
LIN {X 0.067,Y -437.332,Z 702.836,A 0.000,B 0.000,C 90.000,E1 6.486} C_DIS
LIN {X 0.142,Y -441.132,Z 702.821,A 0.000,B 0.000,C 90.000,E1 3.841} C_DIS
LIN {X 0.154,Y -444.768,Z 702.809,A 0.000,B 0.000,C 90.000,E1 1.547} C_DIS
LIN {X -0.131,Y -448.462,Z 702.797,A 0.000,B 0.000,C 90.000,E1 359.484} C_DIS
LIN {X 0.203,Y -451.522,Z 702.788,A 0.000,B 0.000,C 90.000,E1 357.822} C_DIS
LIN {X -0.107,Y -455.337,Z 702.777,A 0.000,B 0.000,C 90.000,E1 355.927} C_DIS
LIN {X -0.116,Y -459.864,Z 702.765,A 0.000,B 0.000,C 90.000,E1 353.685} C_DIS
LIN {X 0.111,Y -463.047,Z 702.756,A 0.000,B 0.000,C 90.000,E1 352.064} C_DIS
LIN {X -0.055,Y -466.121,Z 702.747,A 0.000,B 0.000,C 90.000,E1 350.500} C_DIS
LIN {X 0.191,Y -469.666,Z 702.737,A 0.000,B 0.000,C 90.000,E1 348.578} C_DIS
LIN {X -0.068,Y -471.926,Z 702.730,A 0.000,B 0.000,C 90.000,E1 347.353} C_DIS
LIN {X 0.044,Y -475.346,Z 702.719,A 0.000,B 0.000,C 90.000,E1 345.463} C_DIS
LIN {X -0.097,Y -478.829,Z 702.709,A 0.000,B 0.000,C 90.000,E1 343.614} C_DIS
LIN {X -0.161,Y -482.483,Z 702.699,A 0.000,B 0.000,C 90.000,E1 341.764} C_DIS
LIN {X 0.144,Y -485.666,Z 702.690,A 0.000,B 0.000,C 90.000,E1 340.188} C_DIS
LIN {X 0.127,Y -490.866,Z 702.676,A 0.000,B 0.000,C 90.000,E1 337.741} C_DIS
LIN {X 0.173,Y -492.997,Z 702.672,A 0.000,B 0.000,C 90.000,E1 336.975} C_DIS
LIN {X -0.035,Y -493.475,Z 702.671,A 0.000,B 0.000,C 90.000,E1 336.847} C_DIS
LIN {X -0.058,Y -494.981,Z 702.669,A 0.000,B 0.000,C 90.000,E1 336.485} C_DIS
LIN {X 0.115,Y -496.909,Z 702.667,A 0.000,B 0.000,C 90.000,E1 336.125} C_DIS
LIN {X -0.086,Y -499.081,Z 702.666,A 0.000,B 0.000,C 90.000,E1 335.845} C_DIS
LIN {X 0.173,Y -500.324,Z 702.665,A 0.000,B 0.000,C 90.000,E1 335.665} C_DIS
LIN {X 0.032,Y -504.623,Z 702.663,A 0.000,B 0.000,C 90.000,E1 335.281} C_DIS
LIN {X -0.092,Y -510.331,Z 702.660,A 0.000,B 0.000,C 90.000,E1 334.845} C_DIS
LIN {X -0.282,Y -528.555,Z 702.653,A 0.000,B 0.000,C 90.000,E1 333.640} C_DIS
LIN {X 0.105,Y -536.257,Z 702.651,A 0.000,B 0.000,C 90.000,E1 333.076} C_DIS
LIN {X 0.228,Y -540.728,Z 702.649,A 0.000,B 0.000,C 90.000,E1 332.743} C_DIS
LIN {X -0.200,Y -547.908,Z 702.646,A 0.000,B 0.000,C 90.000,E1 332.231} C_DIS
LIN {X 0.155,Y -552.161,Z 702.644,A 0.000,B 0.000,C 90.000,E1 331.847} C_DIS
LIN {X -0.100,Y -557.645,Z 702.641,A 0.000,B 0.000,C 90.000,E1 331.385} C_DIS
LIN {X -0.025,Y -562.951,Z 702.638,A 0.000,B 0.000,C 90.000,E1 330.873} C_DIS
LIN {X 0.102,Y -570.765,Z 702.634,A 0.000,B 0.000,C 90.000,E1 330.078} C_DIS
LIN {X 0.088,Y -578.207,Z 702.629,A 0.000,B 0.000,C 90.000,E1 329.282} C_DIS
LIN {X -0.012,Y -585.502,Z 702.625,A 0.000,B 0.000,C 90.000,E1 328.486} C_DIS
LIN {X 0.253,Y -592.670,Z 702.621,A 0.000,B 0.000,C 90.000,E1 327.661} C_DIS
LIN {X 0.027,Y -600.584,Z 702.615,A 0.000,B 0.000,C 90.000,E1 326.755} C_DIS
LIN {X 0.139,Y -605.865,Z 702.612,A 0.000,B 0.000,C 90.000,E1 326.087} C_DIS
LIN {X 0.099,Y -611.881,Z 702.607,A 0.000,B 0.000,C 90.000,E1 325.308} C_DIS
LIN {X -0.204,Y -616.544,Z 702.604,A 0.000,B 0.000,C 90.000,E1 324.689} C_DIS
LIN {X -0.155,Y -622.760,Z 702.599,A 0.000,B 0.000,C 90.000,E1 323.783} C_DIS
LIN {X -0.025,Y -627.728,Z 702.594,A 0.000,B 0.000,C 90.000,E1 323.004} C_DIS
LIN {X 0.021,Y -633.873,Z 702.589,A 0.000,B 0.000,C 90.000,E1 321.984} C_DIS
LIN {X -0.238,Y -638.302,Z 702.585,A 0.000,B 0.000,C 90.000,E1 321.251} C_DIS
LIN {X -0.050,Y -643.239,Z 702.580,A 0.000,B 0.000,C 90.000,E1 320.356} C_DIS
LIN {X 0.129,Y -649.241,Z 702.574,A 0.000,B 0.000,C 90.000,E1 319.218} C_DIS
LIN {X 0.402,Y -654.937,Z 702.567,A 0.000,B 0.000,C 90.000,E1 318.081} C_DIS
LIN {X 0.295,Y -659.073,Z 702.563,A 0.000,B 0.000,C 90.000,E1 317.229} C_DIS
LIN {X -0.233,Y -662.332,Z 702.558,A 0.000,B 0.000,C 90.000,E1 316.539} C_DIS
LIN {X -0.282,Y -666.454,Z 702.553,A 0.000,B 0.000,C 90.000,E1 315.567} C_DIS
LIN {X -0.275,Y -670.220,Z 702.548,A 0.000,B 0.000,C 90.000,E1 314.595} C_DIS
LIN {X -0.201,Y -674.655,Z 702.541,A 0.000,B 0.000,C 90.000,E1 313.380} C_DIS
LIN {X -0.025,Y -678.930,Z 702.534,A 0.000,B 0.000,C 90.000,E1 312.162} C_DIS
LIN {X -0.325,Y -682.152,Z 702.529,A 0.000,B 0.000,C 90.000,E1 311.229} C_DIS
LIN {X -0.073,Y -685.109,Z 702.524,A 0.000,B 0.000,C 90.000,E1 310.253} C_DIS
LIN {X -0.363,Y -687.114,Z 702.520,A 0.000,B 0.000,C 90.000,E1 309.564} C_DIS
LIN {X -0.105,Y -688.956,Z 702.516,A 0.000,B 0.000,C 90.000,E1 308.830} C_DIS
LIN {X 0.115,Y -690.139,Z 702.513,A 0.000,B 0.000,C 90.000,E1 308.338} C_DIS
LIN {X 0.100,Y -692.571,Z 702.507,A 0.000,B 0.000,C 90.000,E1 307.156} C_DIS
LIN {X -0.305,Y -694.687,Z 702.500,A 0.000,B 0.000,C 90.000,E1 306.011} C_DIS
LIN {X -0.390,Y -695.834,Z 702.496,A 0.000,B 0.000,C 90.000,E1 305.311} C_DIS
LIN {X -0.184,Y -697.432,Z 702.490,A 0.000,B 0.000,C 90.000,E1 304.119} C_DIS
LIN {X -0.003,Y -698.525,Z 702.484,A 0.000,B 0.000,C 90.000,E1 303.166} C_DIS
LIN {X 0.194,Y -699.379,Z 702.479,A 0.000,B 0.000,C 90.000,E1 302.212} C_DIS
LIN {X 0.061,Y -700.426,Z 702.473,A 0.000,B 0.000,C 90.000,E1 301.052} C_DIS
LIN {X 0.252,Y -700.928,Z 702.469,A 0.000,B 0.000,C 90.000,E1 300.335} C_DIS
LIN {X 0.050,Y -701.500,Z 702.461,A 0.000,B 0.000,C 90.000,E1 298.949} C_DIS
LIN {X -0.154,Y -702.024,Z 702.453,A 0.000,B 0.000,C 90.000,E1 297.564} C_DIS
LIN {X 0.196,Y -703.020,Z 702.443,A 0.000,B 0.000,C 90.000,E1 295.668} C_DIS
LIN {X 0.124,Y -703.063,Z 702.440,A 0.000,B 0.000,C 90.000,E1 295.207} C_DIS
LIN {X 0.107,Y -702.909,Z 702.439,A 0.000,B 0.000,C 90.000,E1 294.975} C_DIS
LIN {X 0.031,Y -702.155,Z 702.436,A 0.000,B 0.000,C 90.000,E1 294.515} C_DIS
LIN {X 0.307,Y -701.277,Z 702.435,A 0.000,B 0.000,C 90.000,E1 294.259} C_DIS
LIN {X -0.074,Y -698.225,Z 702.432,A 0.000,B 0.000,C 90.000,E1 293.823} C_DIS
LIN {X 0.058,Y -697.280,Z 702.432,A 0.000,B 0.000,C 90.000,E1 293.695} C_DIS
LIN {X -0.090,Y -695.870,Z 702.431,A 0.000,B 0.000,C 90.000,E1 293.590} C_DIS
LIN {X 0.155,Y -694.008,Z 702.430,A 0.000,B 0.000,C 90.000,E1 293.462} C_DIS
LIN {X 0.035,Y -688.493,Z 702.429,A 0.000,B 0.000,C 90.000,E1 293.206} C_DIS
LIN {X 0.034,Y -686.542,Z 702.429,A 0.000,B 0.000,C 90.000,E1 293.131} C_DIS
LIN {X 0.319,Y -679.470,Z 702.428,A 0.000,B 0.000,C 90.000,E1 292.950} C_DIS
LIN {X -0.126,Y -677.468,Z 702.427,A 0.000,B 0.000,C 90.000,E1 292.950} C_DIS
LIN {X -0.015,Y -663.338,Z 702.427,A 0.000,B 0.000,C 90.000,E1 292.770} C_DIS
LIN {X -0.140,Y -646.091,Z 702.425,A 0.000,B 0.000,C 90.000,E1 292.514} C_DIS
LIN {X -0.221,Y -636.246,Z 702.424,A 0.000,B 0.000,C 90.000,E1 292.333} C_DIS
LIN {X 0.107,Y -626.258,Z 702.423,A 0.000,B 0.000,C 90.000,E1 292.078} C_DIS
LIN {X -0.200,Y -609.418,Z 702.420,A 0.000,B 0.000,C 90.000,E1 291.663} C_DIS
LIN {X -0.049,Y -574.741,Z 702.415,A 0.000,B 0.000,C 90.000,E1 290.610} C_DIS
LIN {X 0.267,Y -569.228,Z 702.414,A 0.000,B 0.000,C 90.000,E1 290.429} C_DIS
LIN {X -0.343,Y -562.469,Z 702.412,A 0.000,B 0.000,C 90.000,E1 290.248} C_DIS
LIN {X -0.198,Y -558.716,Z 702.411,A 0.000,B 0.000,C 90.000,E1 290.066} C_DIS
LIN {X 0.198,Y -556.057,Z 702.410,A 0.000,B 0.000,C 90.000,E1 289.812} C_DIS
LIN {X 0.162,Y -556.036,Z 702.410,A 0.000,B 0.000,C 90.000,E1 289.812} C_DIS
LIN {X -0.034,Y -555.181,Z 702.409,A 0.000,B 0.000,C 90.000,E1 289.631} C_DIS
LIN {X -0.016,Y -554.521,Z 702.406,A 0.000,B 0.000,C 90.000,E1 289.141} C_DIS
LIN {X -0.190,Y -554.014,Z 702.399,A 0.000,B 0.000,C 90.000,E1 287.764} C_DIS
LIN {X -0.094,Y -553.358,Z 702.389,A 0.000,B 0.000,C 90.000,E1 286.079} C_DIS
LIN {X -0.062,Y -552.671,Z 702.378,A 0.000,B 0.000,C 90.000,E1 284.120} C_DIS
LIN {X -0.006,Y -552.142,Z 702.371,A 0.000,B 0.000,C 90.000,E1 282.715} C_DIS
LIN {X -0.254,Y -551.309,Z 702.360,A 0.000,B 0.000,C 90.000,E1 280.782} C_DIS
LIN {X 0.128,Y -550.192,Z 702.346,A 0.000,B 0.000,C 90.000,E1 278.219} C_DIS
LIN {X 0.097,Y -549.468,Z 702.335,A 0.000,B 0.000,C 90.000,E1 276.258} C_DIS
LIN {X -0.001,Y -549.076,Z 702.324,A 0.000,B 0.000,C 90.000,E1 274.302} C_DIS
LIN {X 0.226,Y -548.951,Z 702.318,A 0.000,B 0.000,C 90.000,E1 273.154} C_DIS
LIN {X 0.021,Y -548.422,Z 702.308,A 0.000,B 0.000,C 90.000,E1 271.489} C_DIS
LIN {X 0.169,Y -548.112,Z 702.304,A 0.000,B 0.000,C 90.000,E1 270.630} C_DIS
LIN {X -0.091,Y -547.109,Z 702.294,A 0.000,B 0.000,C 90.000,E1 268.969} C_DIS
LIN {X 0.221,Y -545.907,Z 702.283,A 0.000,B 0.000,C 90.000,E1 266.963} C_DIS
LIN {X -0.053,Y -544.780,Z 702.274,A 0.000,B 0.000,C 90.000,E1 265.298} C_DIS
LIN {X -0.225,Y -543.296,Z 702.263,A 0.000,B 0.000,C 90.000,E1 263.337} C_DIS
LIN {X 0.026,Y -541.989,Z 702.255,A 0.000,B 0.000,C 90.000,E1 261.894} C_DIS
LIN {X -0.148,Y -540.117,Z 702.244,A 0.000,B 0.000,C 90.000,E1 259.926} C_DIS
LIN {X -0.249,Y -538.492,Z 702.234,A 0.000,B 0.000,C 90.000,E1 258.229} C_DIS
LIN {X 0.200,Y -537.251,Z 702.227,A 0.000,B 0.000,C 90.000,E1 256.756} C_DIS
LIN {X 0.108,Y -535.980,Z 702.219,A 0.000,B 0.000,C 90.000,E1 255.338} C_DIS
LIN {X -0.060,Y -534.873,Z 702.212,A 0.000,B 0.000,C 90.000,E1 254.212} C_DIS
LIN {X -0.024,Y -533.058,Z 702.203,A 0.000,B 0.000,C 90.000,E1 252.489} C_DIS
LIN {X 0.098,Y -531.684,Z 702.195,A 0.000,B 0.000,C 90.000,E1 251.040} C_DIS
LIN {X 0.182,Y -530.349,Z 702.188,A 0.000,B 0.000,C 90.000,E1 249.880} C_DIS
LIN {X -0.061,Y -528.450,Z 702.180,A 0.000,B 0.000,C 90.000,E1 248.465} C_DIS
LIN {X 0.146,Y -526.361,Z 702.172,A 0.000,B 0.000,C 90.000,E1 246.997} C_DIS
LIN {X -0.307,Y -525.128,Z 702.168,A 0.000,B 0.000,C 90.000,E1 246.177} C_DIS
LIN {X -0.074,Y -522.225,Z 702.158,A 0.000,B 0.000,C 90.000,E1 244.409} C_DIS
LIN {X -0.014,Y -521.228,Z 702.155,A 0.000,B 0.000,C 90.000,E1 243.819} C_DIS
LIN {X -0.096,Y -517.918,Z 702.145,A 0.000,B 0.000,C 90.000,E1 242.076} C_DIS
LIN {X 0.084,Y -515.028,Z 702.137,A 0.000,B 0.000,C 90.000,E1 240.589} C_DIS
LIN {X 0.100,Y -512.542,Z 702.130,A 0.000,B 0.000,C 90.000,E1 239.410} C_DIS
LIN {X -0.126,Y -508.787,Z 702.120,A 0.000,B 0.000,C 90.000,E1 237.661} C_DIS
LIN {X -0.160,Y -504.917,Z 702.110,A 0.000,B 0.000,C 90.000,E1 235.881} C_DIS
LIN {X -0.002,Y -500.955,Z 702.100,A 0.000,B 0.000,C 90.000,E1 234.069} C_DIS
LIN {X -0.064,Y -498.756,Z 702.095,A 0.000,B 0.000,C 90.000,E1 233.176} C_DIS
LIN {X -0.148,Y -494.056,Z 702.085,A 0.000,B 0.000,C 90.000,E1 231.376} C_DIS
LIN {X 0.118,Y -488.929,Z 702.074,A 0.000,B 0.000,C 90.000,E1 229.218} C_DIS
LIN {X 0.003,Y -483.288,Z 702.060,A 0.000,B 0.000,C 90.000,E1 226.782} C_DIS
LIN {X -0.012,Y -479.836,Z 702.051,A 0.000,B 0.000,C 90.000,E1 225.243} C_DIS
LIN {X -0.203,Y -477.090,Z 702.044,A 0.000,B 0.000,C 90.000,E1 224.028} C_DIS
LIN {X -0.030,Y -471.613,Z 702.031,A 0.000,B 0.000,C 90.000,E1 221.515} C_DIS
LIN {X -0.127,Y -467.504,Z 702.020,A 0.000,B 0.000,C 90.000,E1 219.644} C_DIS
LIN {X -0.122,Y -464.892,Z 702.013,A 0.000,B 0.000,C 90.000,E1 218.382} C_DIS
LIN {X 0.072,Y -460.792,Z 702.003,A 0.000,B 0.000,C 90.000,E1 216.457} C_DIS
LIN {X 0.005,Y -455.826,Z 701.988,A 0.000,B 0.000,C 90.000,E1 213.913} C_DIS
LIN {X -0.153,Y -452.128,Z 701.978,A 0.000,B 0.000,C 90.000,E1 212.005} C_DIS
LIN {X -0.089,Y -447.260,Z 701.963,A 0.000,B 0.000,C 90.000,E1 209.411} C_DIS
LIN {X -0.117,Y -443.792,Z 701.953,A 0.000,B 0.000,C 90.000,E1 207.462} C_DIS
LIN {X 0.123,Y -440.751,Z 701.943,A 0.000,B 0.000,C 90.000,E1 205.796} C_DIS
LIN {X 0.130,Y -437.174,Z 701.932,A 0.000,B 0.000,C 90.000,E1 203.823} C_DIS
LIN {X -0.135,Y -434.148,Z 701.923,A 0.000,B 0.000,C 90.000,E1 202.206} C_DIS
LIN {X -0.030,Y -431.764,Z 701.916,A 0.000,B 0.000,C 90.000,E1 200.865} C_DIS
LIN {X 0.065,Y -428.142,Z 701.905,A 0.000,B 0.000,C 90.000,E1 198.852} C_DIS
LIN {X 0.069,Y -425.653,Z 701.897,A 0.000,B 0.000,C 90.000,E1 197.511} C_DIS
LIN {X -0.035,Y -422.619,Z 701.888,A 0.000,B 0.000,C 90.000,E1 195.843} C_DIS
LIN {X -0.139,Y -418.943,Z 701.877,A 0.000,B 0.000,C 90.000,E1 193.828} C_DIS
LIN {X -0.075,Y -416.039,Z 701.867,A 0.000,B 0.000,C 90.000,E1 192.119} C_DIS
LIN {X -0.122,Y -412.553,Z 701.856,A 0.000,B 0.000,C 90.000,E1 190.074} C_DIS
LIN {X 0.067,Y -408.158,Z 701.841,A 0.000,B 0.000,C 90.000,E1 187.296} C_DIS
LIN {X 0.052,Y -405.123,Z 701.829,A 0.000,B 0.000,C 90.000,E1 185.220} C_DIS
LIN {X -0.098,Y -402.163,Z 701.818,A 0.000,B 0.000,C 90.000,E1 183.154} C_DIS
LIN {X -0.061,Y -398.428,Z 701.800,A 0.000,B 0.000,C 90.000,E1 180.000} C_DIS
LIN {X -0.153,Y -395.413,Z 701.782,A 0.000,B 0.000,C 90.000,E1 176.846} C_DIS
LIN {X -0.179,Y -392.258,Z 701.755,A 0.000,B 0.000,C 90.000,E1 171.894} C_DIS
LIN {X -0.015,Y -391.567,Z 701.745,A 0.000,B 0.000,C 90.000,E1 170.095} C_DIS
LIN {X 0.155,Y -390.985,Z 701.733,A 0.000,B 0.000,C 90.000,E1 167.937} C_DIS
LIN {X 0.000,Y -390.359,Z 701.721,A 0.000,B 0.000,C 90.000,E1 165.825} C_DIS
LIN {X 0.020,Y -389.946,Z 701.709,A 0.000,B 0.000,C 90.000,E1 163.685} C_DIS
LIN {X -0.151,Y -389.750,Z 701.694,A 0.000,B 0.000,C 90.000,E1 160.859} C_DIS
LIN {X -0.152,Y -389.766,Z 701.682,A 0.000,B 0.000,C 90.000,E1 158.720} C_DIS
LIN {X 0.171,Y -389.913,Z 701.668,A 0.000,B 0.000,C 90.000,E1 156.177} C_DIS
LIN {X -0.060,Y -390.225,Z 701.654,A 0.000,B 0.000,C 90.000,E1 153.717} C_DIS
LIN {X 0.051,Y -390.502,Z 701.642,A 0.000,B 0.000,C 90.000,E1 151.563} C_DIS
LIN {X 0.120,Y -391.544,Z 701.622,A 0.000,B 0.000,C 90.000,E1 147.995} C_DIS
LIN {X -0.141,Y -393.490,Z 701.603,A 0.000,B 0.000,C 90.000,E1 144.482} C_DIS
LIN {X 0.093,Y -395.848,Z 701.587,A 0.000,B 0.000,C 90.000,E1 141.618} C_DIS
LIN {X -0.077,Y -398.356,Z 701.573,A 0.000,B 0.000,C 90.000,E1 139.175} C_DIS
LIN {X 0.045,Y -401.567,Z 701.560,A 0.000,B 0.000,C 90.000,E1 136.701} C_DIS
LIN {X 0.254,Y -402.927,Z 701.556,A 0.000,B 0.000,C 90.000,E1 135.972} C_DIS
LIN {X 0.001,Y -405.097,Z 701.552,A 0.000,B 0.000,C 90.000,E1 135.324} C_DIS
LIN {X -0.112,Y -406.862,Z 701.550,A 0.000,B 0.000,C 90.000,E1 135.000} C_DIS
LIN {X -0.195,Y -407.649,Z 701.549,A 0.000,B 0.000,C 90.000,E1 134.838} C_DIS
LIN {X 0.225,Y -410.246,Z 701.547,A 0.000,B 0.000,C 90.000,E1 134.433} C_DIS
LIN {X 0.149,Y -411.421,Z 701.546,A 0.000,B 0.000,C 90.000,E1 134.271} C_DIS
LIN {X 0.143,Y -415.819,Z 701.543,A 0.000,B 0.000,C 90.000,E1 133.785} C_DIS
LIN {X -0.119,Y -421.424,Z 701.540,A 0.000,B 0.000,C 90.000,E1 133.257} C_DIS
LIN {X -0.153,Y -433.213,Z 701.534,A 0.000,B 0.000,C 90.000,E1 132.162} C_DIS
LIN {X 0.009,Y -448.426,Z 701.527,A 0.000,B 0.000,C 90.000,E1 130.825} C_DIS
LIN {X -0.221,Y -457.452,Z 701.523,A 0.000,B 0.000,C 90.000,E1 130.092} C_DIS
LIN {X -0.211,Y -467.802,Z 701.518,A 0.000,B 0.000,C 90.000,E1 129.197} C_DIS
LIN {X -0.238,Y -475.145,Z 701.514,A 0.000,B 0.000,C 90.000,E1 128.543} C_DIS
LIN {X -0.189,Y -483.712,Z 701.510,A 0.000,B 0.000,C 90.000,E1 127.729} C_DIS
LIN {X 0.280,Y -491.934,Z 701.505,A 0.000,B 0.000,C 90.000,E1 126.870} C_DIS
LIN {X -0.016,Y -498.655,Z 701.501,A 0.000,B 0.000,C 90.000,E1 126.217} C_DIS
LIN {X -0.138,Y -505.295,Z 701.497,A 0.000,B 0.000,C 90.000,E1 125.518} C_DIS
LIN {X -0.255,Y -511.323,Z 701.493,A 0.000,B 0.000,C 90.000,E1 124.818} C_DIS
LIN {X -0.324,Y -514.762,Z 701.491,A 0.000,B 0.000,C 90.000,E1 124.405} C_DIS
LIN {X -0.075,Y -518.937,Z 701.488,A 0.000,B 0.000,C 90.000,E1 123.833} C_DIS
LIN {X 0.120,Y -522.988,Z 701.485,A 0.000,B 0.000,C 90.000,E1 123.245} C_DIS
LIN {X 0.113,Y -526.760,Z 701.482,A 0.000,B 0.000,C 90.000,E1 122.673} C_DIS
LIN {X -0.216,Y -531.118,Z 701.478,A 0.000,B 0.000,C 90.000,E1 122.005} C_DIS
LIN {X 0.039,Y -535.107,Z 701.474,A 0.000,B 0.000,C 90.000,E1 121.258} C_DIS
LIN {X 0.057,Y -538.723,Z 701.470,A 0.000,B 0.000,C 90.000,E1 120.541} C_DIS
LIN {X 0.252,Y -542.635,Z 701.465,A 0.000,B 0.000,C 90.000,E1 119.667} C_DIS
LIN {X 0.219,Y -546.355,Z 701.460,A 0.000,B 0.000,C 90.000,E1 118.821} C_DIS
LIN {X -0.137,Y -549.299,Z 701.456,A 0.000,B 0.000,C 90.000,E1 118.153} C_DIS
LIN {X -0.110,Y -552.608,Z 701.452,A 0.000,B 0.000,C 90.000,E1 117.308} C_DIS
LIN {X -0.299,Y -555.686,Z 701.447,A 0.000,B 0.000,C 90.000,E1 116.488} C_DIS
LIN {X 0.296,Y -558.609,Z 701.442,A 0.000,B 0.000,C 90.000,E1 115.591} C_DIS
LIN {X 0.178,Y -561.219,Z 701.438,A 0.000,B 0.000,C 90.000,E1 114.771} C_DIS
LIN {X 0.088,Y -563.570,Z 701.433,A 0.000,B 0.000,C 90.000,E1 113.951} C_DIS
LIN {X 0.019,Y -565.675,Z 701.429,A 0.000,B 0.000,C 90.000,E1 113.131} C_DIS
LIN {X -0.252,Y -567.480,Z 701.424,A 0.000,B 0.000,C 90.000,E1 112.333} C_DIS
LIN {X 0.192,Y -570.027,Z 701.416,A 0.000,B 0.000,C 90.000,E1 110.918} C_DIS
LIN {X -0.051,Y -572.433,Z 701.409,A 0.000,B 0.000,C 90.000,E1 109.577} C_DIS
LIN {X -0.077,Y -575.186,Z 701.400,A 0.000,B 0.000,C 90.000,E1 107.946} C_DIS
LIN {X 0.136,Y -577.420,Z 701.392,A 0.000,B 0.000,C 90.000,E1 106.567} C_DIS
LIN {X -0.176,Y -579.447,Z 701.385,A 0.000,B 0.000,C 90.000,E1 105.245} C_DIS
LIN {X 0.173,Y -581.895,Z 701.376,A 0.000,B 0.000,C 90.000,E1 103.592} C_DIS
LIN {X 0.206,Y -583.896,Z 701.368,A 0.000,B 0.000,C 90.000,E1 102.243} C_DIS
LIN {X -0.240,Y -587.115,Z 701.356,A 0.000,B 0.000,C 90.000,E1 100.141} C_DIS
LIN {X 0.192,Y -588.604,Z 701.350,A 0.000,B 0.000,C 90.000,E1 99.029} C_DIS
LIN {X 0.135,Y -590.284,Z 701.343,A 0.000,B 0.000,C 90.000,E1 97.701} C_DIS
LIN {X -0.150,Y -591.607,Z 701.337,A 0.000,B 0.000,C 90.000,E1 96.663} C_DIS
LIN {X 0.046,Y -593.494,Z 701.328,A 0.000,B 0.000,C 90.000,E1 95.049} C_DIS
LIN {X 0.012,Y -594.957,Z 701.321,A 0.000,B 0.000,C 90.000,E1 93.726} C_DIS
LIN {X -0.262,Y -595.966,Z 701.315,A 0.000,B 0.000,C 90.000,E1 92.694} C_DIS
LIN {X 0.300,Y -597.163,Z 701.308,A 0.000,B 0.000,C 90.000,E1 91.318} C_DIS
LIN {X 0.273,Y -598.040,Z 701.300,A 0.000,B 0.000,C 90.000,E1 90.000} C_DIS
LIN {X 0.023,Y -598.560,Z 701.294,A 0.000,B 0.000,C 90.000,E1 88.969} C_DIS
LIN {X 0.270,Y -599.068,Z 701.286,A 0.000,B 0.000,C 90.000,E1 87.364} C_DIS
LIN {X -0.312,Y -599.370,Z 701.278,A 0.000,B 0.000,C 90.000,E1 86.102} C_DIS
LIN {X -0.253,Y -599.525,Z 701.271,A 0.000,B 0.000,C 90.000,E1 84.780} C_DIS
LIN {X 0.178,Y -599.510,Z 701.265,A 0.000,B 0.000,C 90.000,E1 83.685} C_DIS
LIN {X 0.307,Y -599.323,Z 701.258,A 0.000,B 0.000,C 90.000,E1 82.356} C_DIS
LIN {X 0.133,Y -599.025,Z 701.252,A 0.000,B 0.000,C 90.000,E1 81.319} C_DIS
LIN {X -0.254,Y -598.366,Z 701.245,A 0.000,B 0.000,C 90.000,E1 80.038} C_DIS
LIN {X -0.062,Y -597.367,Z 701.237,A 0.000,B 0.000,C 90.000,E1 78.701} C_DIS
LIN {X -0.063,Y -596.577,Z 701.231,A 0.000,B 0.000,C 90.000,E1 77.645} C_DIS
LIN {X 0.210,Y -595.386,Z 701.224,A 0.000,B 0.000,C 90.000,E1 76.297} C_DIS
LIN {X -0.275,Y -593.785,Z 701.215,A 0.000,B 0.000,C 90.000,E1 74.755} C_DIS
LIN {X 0.250,Y -592.314,Z 701.208,A 0.000,B 0.000,C 90.000,E1 73.378} C_DIS
LIN {X -0.124,Y -590.367,Z 701.199,A 0.000,B 0.000,C 90.000,E1 71.819} C_DIS
LIN {X 0.096,Y -588.947,Z 701.193,A 0.000,B 0.000,C 90.000,E1 70.732} C_DIS
LIN {X 0.162,Y -586.966,Z 701.186,A 0.000,B 0.000,C 90.000,E1 69.390} C_DIS
LIN {X -0.011,Y -585.253,Z 701.180,A 0.000,B 0.000,C 90.000,E1 68.337} C_DIS
LIN {X -0.074,Y -583.823,Z 701.175,A 0.000,B 0.000,C 90.000,E1 67.539} C_DIS
LIN {X -0.156,Y -582.189,Z 701.171,A 0.000,B 0.000,C 90.000,E1 66.741} C_DIS
LIN {X -0.164,Y -579.938,Z 701.165,A 0.000,B 0.000,C 90.000,E1 65.665} C_DIS
LIN {X -0.055,Y -577.982,Z 701.160,A 0.000,B 0.000,C 90.000,E1 64.845} C_DIS
LIN {X -0.117,Y -575.032,Z 701.154,A 0.000,B 0.000,C 90.000,E1 63.768} C_DIS
LIN {X -0.068,Y -572.676,Z 701.150,A 0.000,B 0.000,C 90.000,E1 62.948} C_DIS
LIN {X 0.214,Y -570.149,Z 701.145,A 0.000,B 0.000,C 90.000,E1 62.103} C_DIS
LIN {X -0.206,Y -566.513,Z 701.139,A 0.000,B 0.000,C 90.000,E1 61.051} C_DIS
LIN {X 0.010,Y -563.494,Z 701.135,A 0.000,B 0.000,C 90.000,E1 60.205} C_DIS
LIN {X -0.296,Y -560.241,Z 701.130,A 0.000,B 0.000,C 90.000,E1 59.410} C_DIS
LIN {X 0.127,Y -556.475,Z 701.125,A 0.000,B 0.000,C 90.000,E1 58.535} C_DIS
LIN {X -0.143,Y -552.985,Z 701.121,A 0.000,B 0.000,C 90.000,E1 57.867} C_DIS
LIN {X -0.146,Y -549.088,Z 701.118,A 0.000,B 0.000,C 90.000,E1 57.168} C_DIS
LIN {X 0.106,Y -545.707,Z 701.114,A 0.000,B 0.000,C 90.000,E1 56.580} C_DIS
LIN {X 0.177,Y -542.006,Z 701.111,A 0.000,B 0.000,C 90.000,E1 56.008} C_DIS
LIN {X -0.081,Y -537.990,Z 701.108,A 0.000,B 0.000,C 90.000,E1 55.468} C_DIS
LIN {X -0.060,Y -533.584,Z 701.105,A 0.000,B 0.000,C 90.000,E1 54.895} C_DIS
LIN {X -0.046,Y -528.621,Z 701.102,A 0.000,B 0.000,C 90.000,E1 54.322} C_DIS
LIN {X 0.132,Y -523.642,Z 701.099,A 0.000,B 0.000,C 90.000,E1 53.783} C_DIS
LIN {X -0.071,Y -518.080,Z 701.096,A 0.000,B 0.000,C 90.000,E1 53.290} C_DIS
LIN {X -0.225,Y -513.355,Z 701.094,A 0.000,B 0.000,C 90.000,E1 52.924} C_DIS
LIN {X -0.063,Y -508.809,Z 701.092,A 0.000,B 0.000,C 90.000,E1 52.557} C_DIS
LIN {X 0.011,Y -502.399,Z 701.090,A 0.000,B 0.000,C 90.000,E1 52.110} C_DIS
LIN {X 0.033,Y -492.639,Z 701.086,A 0.000,B 0.000,C 90.000,E1 51.492} C_DIS
LIN {X 0.036,Y -479.381,Z 701.082,A 0.000,B 0.000,C 90.000,E1 50.723} C_DIS
LIN {X 0.199,Y -463.202,Z 701.077,A 0.000,B 0.000,C 90.000,E1 49.747} C_DIS
LIN {X -0.038,Y -433.994,Z 701.066,A 0.000,B 0.000,C 90.000,E1 47.957} C_DIS
LIN {X 0.091,Y -423.057,Z 701.062,A 0.000,B 0.000,C 90.000,E1 47.148} C_DIS
LIN {X 0.064,Y -423.014,Z 701.062,A 0.000,B 0.000,C 90.000,E1 47.148} C_DIS
LIN {X -0.015,Y -418.392,Z 701.048,A 0.000,B 0.000,C 90.000,E1 44.717} C_DIS
LIN {X 0.082,Y -410.153,Z 701.028,A 0.000,B 0.000,C 90.000,E1 40.943} C_DIS
LIN {X 0.155,Y -410.273,Z 701.012,A 0.000,B 0.000,C 90.000,E1 38.177} C_DIS
LIN {X 0.114,Y -411.390,Z 700.993,A 0.000,B 0.000,C 90.000,E1 34.739} C_DIS
LIN {X 0.048,Y -412.018,Z 700.985,A 0.000,B 0.000,C 90.000,E1 33.372} C_DIS
LIN {X -0.203,Y -413.226,Z 700.972,A 0.000,B 0.000,C 90.000,E1 31.003} C_DIS
LIN {X -0.219,Y -414.312,Z 700.961,A 0.000,B 0.000,C 90.000,E1 28.949} C_DIS
LIN {X 0.012,Y -415.325,Z 700.951,A 0.000,B 0.000,C 90.000,E1 27.206} C_DIS
LIN {X 0.096,Y -417.222,Z 700.936,A 0.000,B 0.000,C 90.000,E1 24.463} C_DIS
LIN {X -0.116,Y -419.510,Z 700.921,A 0.000,B 0.000,C 90.000,E1 21.770} C_DIS
LIN {X -0.115,Y -421.841,Z 700.908,A 0.000,B 0.000,C 90.000,E1 19.396} C_DIS
LIN {X 0.040,Y -423.989,Z 700.896,A 0.000,B 0.000,C 90.000,E1 17.347} C_DIS
LIN {X 0.125,Y -426.260,Z 700.885,A 0.000,B 0.000,C 90.000,E1 15.315} C_DIS
LIN {X 0.053,Y -428.280,Z 700.876,A 0.000,B 0.000,C 90.000,E1 13.647} C_DIS
LIN {X -0.078,Y -430.797,Z 700.865,A 0.000,B 0.000,C 90.000,E1 11.658} C_DIS
LIN {X -0.151,Y -433.385,Z 700.854,A 0.000,B 0.000,C 90.000,E1 9.670} C_DIS
LIN {X -0.050,Y -436.930,Z 700.839,A 0.000,B 0.000,C 90.000,E1 7.004} C_DIS
LIN {X 0.102,Y -439.193,Z 700.830,A 0.000,B 0.000,C 90.000,E1 5.334} C_DIS
LIN {X -0.058,Y -442.127,Z 700.819,A 0.000,B 0.000,C 90.000,E1 3.383} C_DIS
LIN {X -0.015,Y -445.819,Z 700.806,A 0.000,B 0.000,C 90.000,E1 1.088} C_DIS
LIN {X -0.123,Y -450.517,Z 700.792,A 0.000,B 0.000,C 90.000,E1 358.511} C_DIS
LIN {X 0.155,Y -454.860,Z 700.779,A 0.000,B 0.000,C 90.000,E1 356.216} C_DIS
LIN {X 0.183,Y -458.047,Z 700.770,A 0.000,B 0.000,C 90.000,E1 354.609} C_DIS
LIN {X 0.132,Y -460.651,Z 700.763,A 0.000,B 0.000,C 90.000,E1 353.337} C_DIS
LIN {X -0.145,Y -463.795,Z 700.754,A 0.000,B 0.000,C 90.000,E1 351.781} C_DIS
LIN {X -0.034,Y -466.256,Z 700.747,A 0.000,B 0.000,C 90.000,E1 350.500} C_DIS
LIN {X 0.215,Y -469.766,Z 700.737,A 0.000,B 0.000,C 90.000,E1 348.578} C_DIS
LIN {X -0.042,Y -472.043,Z 700.730,A 0.000,B 0.000,C 90.000,E1 347.353} C_DIS
LIN {X 0.072,Y -475.463,Z 700.719,A 0.000,B 0.000,C 90.000,E1 345.463} C_DIS
LIN {X -0.065,Y -478.953,Z 700.709,A 0.000,B 0.000,C 90.000,E1 343.614} C_DIS
LIN {X 0.029,Y -481.991,Z 700.700,A 0.000,B 0.000,C 90.000,E1 342.054} C_DIS
LIN {X 0.181,Y -485.762,Z 700.690,A 0.000,B 0.000,C 90.000,E1 340.188} C_DIS
LIN {X 0.138,Y -490.185,Z 700.678,A 0.000,B 0.000,C 90.000,E1 338.050} C_DIS
LIN {X -0.225,Y -492.375,Z 700.673,A 0.000,B 0.000,C 90.000,E1 337.177} C_DIS
LIN {X 0.044,Y -494.219,Z 700.670,A 0.000,B 0.000,C 90.000,E1 336.538} C_DIS
LIN {X 0.141,Y -495.414,Z 700.668,A 0.000,B 0.000,C 90.000,E1 336.230} C_DIS
LIN {X -0.012,Y -497.947,Z 700.666,A 0.000,B 0.000,C 90.000,E1 335.793} C_DIS
LIN {X 0.044,Y -500.158,Z 700.664,A 0.000,B 0.000,C 90.000,E1 335.485} C_DIS
LIN {X -0.035,Y -504.716,Z 700.661,A 0.000,B 0.000,C 90.000,E1 335.049} C_DIS
LIN {X 0.147,Y -510.939,Z 700.659,A 0.000,B 0.000,C 90.000,E1 334.537} C_DIS
LIN {X 0.038,Y -531.397,Z 700.651,A 0.000,B 0.000,C 90.000,E1 333.179} C_DIS
LIN {X 0.046,Y -540.516,Z 700.648,A 0.000,B 0.000,C 90.000,E1 332.538} C_DIS
LIN {X 0.068,Y -547.740,Z 700.644,A 0.000,B 0.000,C 90.000,E1 331.975} C_DIS
LIN {X -0.004,Y -553.421,Z 700.642,A 0.000,B 0.000,C 90.000,E1 331.513} C_DIS
LIN {X -0.306,Y -560.239,Z 700.638,A 0.000,B 0.000,C 90.000,E1 330.923} C_DIS
LIN {X -0.121,Y -569.389,Z 700.633,A 0.000,B 0.000,C 90.000,E1 329.999} C_DIS
LIN {X -0.118,Y -576.898,Z 700.629,A 0.000,B 0.000,C 90.000,E1 329.203} C_DIS
LIN {X 0.038,Y -585.438,Z 700.624,A 0.000,B 0.000,C 90.000,E1 328.250} C_DIS
LIN {X 0.035,Y -591.504,Z 700.620,A 0.000,B 0.000,C 90.000,E1 327.582} C_DIS
LIN {X 0.302,Y -599.522,Z 700.615,A 0.000,B 0.000,C 90.000,E1 326.628} C_DIS
LIN {X -0.139,Y -605.934,Z 700.610,A 0.000,B 0.000,C 90.000,E1 325.881} C_DIS
LIN {X -0.180,Y -611.957,Z 700.606,A 0.000,B 0.000,C 90.000,E1 325.102} C_DIS
LIN {X -0.155,Y -617.563,Z 700.602,A 0.000,B 0.000,C 90.000,E1 324.322} C_DIS
LIN {X -0.091,Y -623.701,Z 700.597,A 0.000,B 0.000,C 90.000,E1 323.417} C_DIS
LIN {X 0.066,Y -627.816,Z 700.593,A 0.000,B 0.000,C 90.000,E1 322.763} C_DIS
LIN {X 0.120,Y -634.021,Z 700.588,A 0.000,B 0.000,C 90.000,E1 321.743} C_DIS
LIN {X 0.372,Y -637.707,Z 700.584,A 0.000,B 0.000,C 90.000,E1 321.090} C_DIS
LIN {X 0.149,Y -642.703,Z 700.579,A 0.000,B 0.000,C 90.000,E1 320.231} C_DIS
LIN {X -0.106,Y -648.119,Z 700.574,A 0.000,B 0.000,C 90.000,E1 319.256} C_DIS
LIN {X -0.348,Y -653.904,Z 700.567,A 0.000,B 0.000,C 90.000,E1 318.162} C_DIS
LIN {X 0.010,Y -658.117,Z 700.563,A 0.000,B 0.000,C 90.000,E1 317.268} C_DIS
LIN {X -0.076,Y -661.453,Z 700.559,A 0.000,B 0.000,C 90.000,E1 316.539} C_DIS
LIN {X -0.136,Y -665.692,Z 700.553,A 0.000,B 0.000,C 90.000,E1 315.567} C_DIS
LIN {X -0.137,Y -669.502,Z 700.548,A 0.000,B 0.000,C 90.000,E1 314.595} C_DIS
LIN {X -0.075,Y -674.013,Z 700.541,A 0.000,B 0.000,C 90.000,E1 313.380} C_DIS
LIN {X 0.092,Y -678.360,Z 700.534,A 0.000,B 0.000,C 90.000,E1 312.162} C_DIS
LIN {X 0.197,Y -680.905,Z 700.530,A 0.000,B 0.000,C 90.000,E1 311.434} C_DIS
LIN {X 0.032,Y -684.700,Z 700.524,A 0.000,B 0.000,C 90.000,E1 310.253} C_DIS
LIN {X -0.261,Y -686.768,Z 700.520,A 0.000,B 0.000,C 90.000,E1 309.564} C_DIS
LIN {X -0.007,Y -688.665,Z 700.516,A 0.000,B 0.000,C 90.000,E1 308.830} C_DIS
LIN {X -0.330,Y -689.865,Z 700.513,A 0.000,B 0.000,C 90.000,E1 308.382} C_DIS
LIN {X 0.191,Y -692.331,Z 700.507,A 0.000,B 0.000,C 90.000,E1 307.156} C_DIS
LIN {X 0.139,Y -694.101,Z 700.501,A 0.000,B 0.000,C 90.000,E1 306.217} C_DIS
LIN {X -0.302,Y -695.729,Z 700.496,A 0.000,B 0.000,C 90.000,E1 305.311} C_DIS
LIN {X -0.098,Y -697.355,Z 700.490,A 0.000,B 0.000,C 90.000,E1 304.119} C_DIS
LIN {X 0.082,Y -698.480,Z 700.484,A 0.000,B 0.000,C 90.000,E1 303.166} C_DIS
LIN {X 0.028,Y -699.156,Z 700.480,A 0.000,B 0.000,C 90.000,E1 302.467} C_DIS
LIN {X 0.121,Y -700.207,Z 700.474,A 0.000,B 0.000,C 90.000,E1 301.288} C_DIS
LIN {X 0.337,Y -700.949,Z 700.469,A 0.000,B 0.000,C 90.000,E1 300.335} C_DIS
LIN {X 0.135,Y -701.551,Z 700.461,A 0.000,B 0.000,C 90.000,E1 298.949} C_DIS
LIN {X -0.113,Y -702.200,Z 700.452,A 0.000,B 0.000,C 90.000,E1 297.334} C_DIS
LIN {X -0.349,Y -703.108,Z 700.443,A 0.000,B 0.000,C 90.000,E1 295.720} C_DIS
LIN {X 0.213,Y -703.147,Z 700.440,A 0.000,B 0.000,C 90.000,E1 295.207} C_DIS
LIN {X 0.197,Y -702.998,Z 700.439,A 0.000,B 0.000,C 90.000,E1 294.975} C_DIS
LIN {X 0.120,Y -702.185,Z 700.436,A 0.000,B 0.000,C 90.000,E1 294.515} C_DIS
LIN {X 0.109,Y -701.328,Z 700.435,A 0.000,B 0.000,C 90.000,E1 294.283} C_DIS
LIN {X 0.016,Y -698.161,Z 700.432,A 0.000,B 0.000,C 90.000,E1 293.823} C_DIS
LIN {X 0.147,Y -697.185,Z 700.432,A 0.000,B 0.000,C 90.000,E1 293.695} C_DIS
LIN {X -0.001,Y -695.789,Z 700.431,A 0.000,B 0.000,C 90.000,E1 293.590} C_DIS
LIN {X 0.237,Y -693.761,Z 700.430,A 0.000,B 0.000,C 90.000,E1 293.462} C_DIS
LIN {X 0.216,Y -688.210,Z 700.429,A 0.000,B 0.000,C 90.000,E1 293.206} C_DIS
LIN {X -0.039,Y -686.131,Z 700.429,A 0.000,B 0.000,C 90.000,E1 293.153} C_DIS
LIN {X -0.101,Y -679.228,Z 700.428,A 0.000,B 0.000,C 90.000,E1 293.003} C_DIS
LIN {X 0.054,Y -676.827,Z 700.428,A 0.000,B 0.000,C 90.000,E1 292.950} C_DIS
LIN {X 0.130,Y -662.645,Z 700.427,A 0.000,B 0.000,C 90.000,E1 292.770} C_DIS
LIN {X 0.009,Y -645.651,Z 700.425,A 0.000,B 0.000,C 90.000,E1 292.514} C_DIS
LIN {X -0.163,Y -635.459,Z 700.424,A 0.000,B 0.000,C 90.000,E1 292.333} C_DIS
LIN {X 0.143,Y -625.550,Z 700.423,A 0.000,B 0.000,C 90.000,E1 292.078} C_DIS
LIN {X -0.201,Y -608.659,Z 700.420,A 0.000,B 0.000,C 90.000,E1 291.663} C_DIS
LIN {X -0.124,Y -575.856,Z 700.415,A 0.000,B 0.000,C 90.000,E1 290.663} C_DIS
LIN {X 0.235,Y -568.507,Z 700.414,A 0.000,B 0.000,C 90.000,E1 290.429} C_DIS
LIN {X -0.279,Y -562.018,Z 700.412,A 0.000,B 0.000,C 90.000,E1 290.248} C_DIS
LIN {X 0.137,Y -558.977,Z 700.412,A 0.000,B 0.000,C 90.000,E1 290.066} C_DIS
LIN {X 0.298,Y -555.980,Z 700.410,A 0.000,B 0.000,C 90.000,E1 289.812} C_DIS
LIN {X 0.263,Y -555.958,Z 700.410,A 0.000,B 0.000,C 90.000,E1 289.812} C_DIS
LIN {X -0.076,Y -555.040,Z 700.409,A 0.000,B 0.000,C 90.000,E1 289.631} C_DIS
LIN {X -0.061,Y -554.462,Z 700.406,A 0.000,B 0.000,C 90.000,E1 289.141} C_DIS
LIN {X -0.234,Y -553.982,Z 700.399,A 0.000,B 0.000,C 90.000,E1 287.764} C_DIS
LIN {X -0.139,Y -553.327,Z 700.389,A 0.000,B 0.000,C 90.000,E1 286.079} C_DIS
LIN {X -0.108,Y -552.639,Z 700.378,A 0.000,B 0.000,C 90.000,E1 284.120} C_DIS
LIN {X -0.051,Y -552.109,Z 700.371,A 0.000,B 0.000,C 90.000,E1 282.715} C_DIS
LIN {X -0.300,Y -551.247,Z 700.360,A 0.000,B 0.000,C 90.000,E1 280.782} C_DIS
LIN {X 0.079,Y -550.154,Z 700.346,A 0.000,B 0.000,C 90.000,E1 278.219} C_DIS
LIN {X 0.047,Y -549.435,Z 700.335,A 0.000,B 0.000,C 90.000,E1 276.258} C_DIS
LIN {X -0.050,Y -549.075,Z 700.324,A 0.000,B 0.000,C 90.000,E1 274.302} C_DIS
LIN {X 0.176,Y -548.958,Z 700.318,A 0.000,B 0.000,C 90.000,E1 273.154} C_DIS
LIN {X -0.077,Y -548.529,Z 700.310,A 0.000,B 0.000,C 90.000,E1 271.776} C_DIS
LIN {X 0.070,Y -548.241,Z 700.305,A 0.000,B 0.000,C 90.000,E1 270.917} C_DIS
LIN {X -0.233,Y -547.484,Z 700.297,A 0.000,B 0.000,C 90.000,E1 269.542} C_DIS
LIN {X 0.095,Y -546.300,Z 700.286,A 0.000,B 0.000,C 90.000,E1 267.535} C_DIS
LIN {X -0.161,Y -545.184,Z 700.277,A 0.000,B 0.000,C 90.000,E1 265.869} C_DIS
LIN {X -0.026,Y -544.555,Z 700.272,A 0.000,B 0.000,C 90.000,E1 265.008} C_DIS
LIN {X 0.269,Y -543.316,Z 700.263,A 0.000,B 0.000,C 90.000,E1 263.280} C_DIS
LIN {X -0.018,Y -541.986,Z 700.255,A 0.000,B 0.000,C 90.000,E1 261.894} C_DIS
LIN {X -0.174,Y -540.361,Z 700.246,A 0.000,B 0.000,C 90.000,E1 260.208} C_DIS
LIN {X 0.164,Y -538.755,Z 700.236,A 0.000,B 0.000,C 90.000,E1 258.465} C_DIS
LIN {X 0.154,Y -537.251,Z 700.227,A 0.000,B 0.000,C 90.000,E1 256.756} C_DIS
LIN {X 0.117,Y -535.736,Z 700.217,A 0.000,B 0.000,C 90.000,E1 255.046} C_DIS
LIN {X 0.135,Y -534.292,Z 700.209,A 0.000,B 0.000,C 90.000,E1 253.614} C_DIS
LIN {X 0.032,Y -531.948,Z 700.196,A 0.000,B 0.000,C 90.000,E1 251.329} C_DIS
LIN {X -0.051,Y -530.731,Z 700.190,A 0.000,B 0.000,C 90.000,E1 250.188} C_DIS
LIN {X 0.019,Y -529.274,Z 700.184,A 0.000,B 0.000,C 90.000,E1 249.028} C_DIS
LIN {X -0.047,Y -527.227,Z 700.176,A 0.000,B 0.000,C 90.000,E1 247.592} C_DIS
LIN {X 0.131,Y -525.149,Z 700.167,A 0.000,B 0.000,C 90.000,E1 246.125} C_DIS
LIN {X -0.115,Y -522.247,Z 700.158,A 0.000,B 0.000,C 90.000,E1 244.409} C_DIS
LIN {X 0.091,Y -520.689,Z 700.153,A 0.000,B 0.000,C 90.000,E1 243.512} C_DIS
LIN {X 0.320,Y -517.914,Z 700.145,A 0.000,B 0.000,C 90.000,E1 242.025} C_DIS
LIN {X 0.043,Y -515.027,Z 700.137,A 0.000,B 0.000,C 90.000,E1 240.589} C_DIS
LIN {X 0.060,Y -512.532,Z 700.130,A 0.000,B 0.000,C 90.000,E1 239.410} C_DIS
LIN {X -0.166,Y -508.777,Z 700.120,A 0.000,B 0.000,C 90.000,E1 237.661} C_DIS
LIN {X -0.200,Y -504.884,Z 700.110,A 0.000,B 0.000,C 90.000,E1 235.881} C_DIS
LIN {X -0.043,Y -500.896,Z 700.100,A 0.000,B 0.000,C 90.000,E1 234.069} C_DIS
LIN {X 0.294,Y -498.724,Z 700.095,A 0.000,B 0.000,C 90.000,E1 233.130} C_DIS
LIN {X 0.197,Y -494.043,Z 700.085,A 0.000,B 0.000,C 90.000,E1 231.331} C_DIS
LIN {X 0.078,Y -488.910,Z 700.074,A 0.000,B 0.000,C 90.000,E1 229.218} C_DIS
LIN {X -0.038,Y -483.265,Z 700.060,A 0.000,B 0.000,C 90.000,E1 226.782} C_DIS
LIN {X 0.072,Y -479.130,Z 700.050,A 0.000,B 0.000,C 90.000,E1 224.919} C_DIS
LIN {X -0.131,Y -476.323,Z 700.043,A 0.000,B 0.000,C 90.000,E1 223.704} C_DIS
LIN {X -0.161,Y -472.242,Z 700.032,A 0.000,B 0.000,C 90.000,E1 221.838} C_DIS
LIN {X -0.169,Y -467.415,Z 700.020,A 0.000,B 0.000,C 90.000,E1 219.644} C_DIS
LIN {X -0.167,Y -464.803,Z 700.013,A 0.000,B 0.000,C 90.000,E1 218.382} C_DIS
LIN {X 0.026,Y -460.734,Z 700.003,A 0.000,B 0.000,C 90.000,E1 216.457} C_DIS
LIN {X -0.041,Y -455.802,Z 699.988,A 0.000,B 0.000,C 90.000,E1 213.913} C_DIS
LIN {X -0.199,Y -452.096,Z 699.978,A 0.000,B 0.000,C 90.000,E1 212.005} C_DIS
LIN {X -0.211,Y -447.839,Z 699.965,A 0.000,B 0.000,C 90.000,E1 209.745} C_DIS
LIN {X -0.016,Y -444.316,Z 699.954,A 0.000,B 0.000,C 90.000,E1 207.769} C_DIS
LIN {X 0.076,Y -440.735,Z 699.943,A 0.000,B 0.000,C 90.000,E1 205.796} C_DIS
LIN {X 0.082,Y -437.156,Z 699.932,A 0.000,B 0.000,C 90.000,E1 203.823} C_DIS
LIN {X -0.182,Y -434.117,Z 699.923,A 0.000,B 0.000,C 90.000,E1 202.206} C_DIS
LIN {X -0.078,Y -431.716,Z 699.916,A 0.000,B 0.000,C 90.000,E1 200.865} C_DIS
LIN {X 0.016,Y -428.090,Z 699.905,A 0.000,B 0.000,C 90.000,E1 198.852} C_DIS
LIN {X 0.020,Y -425.597,Z 699.897,A 0.000,B 0.000,C 90.000,E1 197.511} C_DIS
LIN {X -0.085,Y -422.607,Z 699.888,A 0.000,B 0.000,C 90.000,E1 195.843} C_DIS
LIN {X -0.188,Y -418.952,Z 699.877,A 0.000,B 0.000,C 90.000,E1 193.828} C_DIS
LIN {X -0.124,Y -416.027,Z 699.867,A 0.000,B 0.000,C 90.000,E1 192.119} C_DIS
LIN {X -0.170,Y -412.564,Z 699.856,A 0.000,B 0.000,C 90.000,E1 190.074} C_DIS
LIN {X -0.003,Y -408.699,Z 699.843,A 0.000,B 0.000,C 90.000,E1 187.644} C_DIS
LIN {X 0.001,Y -405.674,Z 699.831,A 0.000,B 0.000,C 90.000,E1 185.568} C_DIS
LIN {X -0.106,Y -402.705,Z 699.819,A 0.000,B 0.000,C 90.000,E1 183.498} C_DIS
LIN {X -0.103,Y -398.518,Z 699.800,A 0.000,B 0.000,C 90.000,E1 180.000} C_DIS
LIN {X 0.204,Y -395.504,Z 699.782,A 0.000,B 0.000,C 90.000,E1 176.788} C_DIS
LIN {X -0.124,Y -392.693,Z 699.759,A 0.000,B 0.000,C 90.000,E1 172.591} C_DIS
LIN {X 0.001,Y -391.850,Z 699.747,A 0.000,B 0.000,C 90.000,E1 170.443} C_DIS
LIN {X 0.128,Y -391.154,Z 699.733,A 0.000,B 0.000,C 90.000,E1 167.937} C_DIS
LIN {X -0.022,Y -390.546,Z 699.721,A 0.000,B 0.000,C 90.000,E1 165.825} C_DIS
LIN {X 0.043,Y -390.096,Z 699.707,A 0.000,B 0.000,C 90.000,E1 163.323} C_DIS
LIN {X -0.201,Y -389.988,Z 699.696,A 0.000,B 0.000,C 90.000,E1 161.221} C_DIS
LIN {X -0.156,Y -390.010,Z 699.682,A 0.000,B 0.000,C 90.000,E1 158.720} C_DIS
LIN {X 0.174,Y -390.165,Z 699.668,A 0.000,B 0.000,C 90.000,E1 156.177} C_DIS
LIN {X -0.050,Y -390.486,Z 699.654,A 0.000,B 0.000,C 90.000,E1 153.717} C_DIS
LIN {X 0.068,Y -390.751,Z 699.642,A 0.000,B 0.000,C 90.000,E1 151.563} C_DIS
LIN {X 0.147,Y -391.803,Z 699.622,A 0.000,B 0.000,C 90.000,E1 147.995} C_DIS
LIN {X -0.106,Y -393.697,Z 699.603,A 0.000,B 0.000,C 90.000,E1 144.482} C_DIS
LIN {X 0.006,Y -394.747,Z 699.595,A 0.000,B 0.000,C 90.000,E1 143.050} C_DIS
LIN {X -0.237,Y -397.715,Z 699.577,A 0.000,B 0.000,C 90.000,E1 139.908} C_DIS
LIN {X 0.168,Y -400.466,Z 699.563,A 0.000,B 0.000,C 90.000,E1 137.391} C_DIS
LIN {X 0.091,Y -401.378,Z 699.560,A 0.000,B 0.000,C 90.000,E1 136.701} C_DIS
LIN {X 0.211,Y -403.038,Z 699.555,A 0.000,B 0.000,C 90.000,E1 135.810} C_DIS
LIN {X -0.050,Y -404.587,Z 699.552,A 0.000,B 0.000,C 90.000,E1 135.324} C_DIS
LIN {X -0.018,Y -406.823,Z 699.549,A 0.000,B 0.000,C 90.000,E1 134.798} C_DIS
LIN {X -0.048,Y -410.267,Z 699.546,A 0.000,B 0.000,C 90.000,E1 134.271} C_DIS
LIN {X 0.181,Y -414.867,Z 699.543,A 0.000,B 0.000,C 90.000,E1 133.704} C_DIS
LIN {X -0.093,Y -420.478,Z 699.540,A 0.000,B 0.000,C 90.000,E1 133.176} C_DIS
LIN {X -0.005,Y -435.796,Z 699.532,A 0.000,B 0.000,C 90.000,E1 131.757} C_DIS
LIN {X 0.226,Y -449.672,Z 699.525,A 0.000,B 0.000,C 90.000,E1 130.539} C_DIS
LIN {X 0.092,Y -457.166,Z 699.522,A 0.000,B 0.000,C 90.000,E1 129.930} C_DIS
LIN {X -0.234,Y -466.315,Z 699.518,A 0.000,B 0.000,C 90.000,E1 129.197} C_DIS
LIN {X 0.014,Y -475.147,Z 699.513,A 0.000,B 0.000,C 90.000,E1 128.382} C_DIS
LIN {X -0.132,Y -482.318,Z 699.510,A 0.000,B 0.000,C 90.000,E1 127.729} C_DIS
LIN {X -0.004,Y -490.605,Z 699.505,A 0.000,B 0.000,C 90.000,E1 126.916} C_DIS
LIN {X 0.052,Y -497.429,Z 699.501,A 0.000,B 0.000,C 90.000,E1 126.217} C_DIS
LIN {X -0.119,Y -502.711,Z 699.498,A 0.000,B 0.000,C 90.000,E1 125.678} C_DIS
LIN {X 0.009,Y -507.702,Z 699.495,A 0.000,B 0.000,C 90.000,E1 125.105} C_DIS
LIN {X 0.025,Y -513.645,Z 699.491,A 0.000,B 0.000,C 90.000,E1 124.405} C_DIS
LIN {X -0.133,Y -518.315,Z 699.488,A 0.000,B 0.000,C 90.000,E1 123.833} C_DIS
LIN {X -0.115,Y -522.585,Z 699.485,A 0.000,B 0.000,C 90.000,E1 123.245} C_DIS
LIN {X 0.066,Y -527.410,Z 699.481,A 0.000,B 0.000,C 90.000,E1 122.498} C_DIS
LIN {X -0.002,Y -531.057,Z 699.477,A 0.000,B 0.000,C 90.000,E1 121.926} C_DIS
LIN {X -0.026,Y -535.112,Z 699.473,A 0.000,B 0.000,C 90.000,E1 121.209} C_DIS
LIN {X 0.270,Y -538.772,Z 699.469,A 0.000,B 0.000,C 90.000,E1 120.463} C_DIS
LIN {X -0.143,Y -542.122,Z 699.466,A 0.000,B 0.000,C 90.000,E1 119.795} C_DIS
LIN {X -0.185,Y -545.910,Z 699.461,A 0.000,B 0.000,C 90.000,E1 118.949} C_DIS
LIN {X -0.184,Y -549.495,Z 699.456,A 0.000,B 0.000,C 90.000,E1 118.103} C_DIS
LIN {X -0.152,Y -552.812,Z 699.451,A 0.000,B 0.000,C 90.000,E1 117.257} C_DIS
LIN {X -0.088,Y -555.893,Z 699.447,A 0.000,B 0.000,C 90.000,E1 116.411} C_DIS
LIN {X -0.238,Y -558.819,Z 699.442,A 0.000,B 0.000,C 90.000,E1 115.591} C_DIS
LIN {X -0.048,Y -562.263,Z 699.436,A 0.000,B 0.000,C 90.000,E1 114.463} C_DIS
LIN {X -0.126,Y -564.534,Z 699.431,A 0.000,B 0.000,C 90.000,E1 113.643} C_DIS
LIN {X 0.005,Y -565.921,Z 699.428,A 0.000,B 0.000,C 90.000,E1 113.078} C_DIS
LIN {X -0.043,Y -567.776,Z 699.424,A 0.000,B 0.000,C 90.000,E1 112.259} C_DIS
LIN {X 0.053,Y -569.845,Z 699.418,A 0.000,B 0.000,C 90.000,E1 111.153} C_DIS
LIN {X -0.201,Y -572.312,Z 699.410,A 0.000,B 0.000,C 90.000,E1 109.812} C_DIS
LIN {X -0.235,Y -575.110,Z 699.401,A 0.000,B 0.000,C 90.000,E1 108.181} C_DIS
LIN {X -0.216,Y -577.825,Z 699.392,A 0.000,B 0.000,C 90.000,E1 106.551} C_DIS
LIN {X -0.126,Y -579.900,Z 699.384,A 0.000,B 0.000,C 90.000,E1 105.190} C_DIS
LIN {X 0.237,Y -582.353,Z 699.375,A 0.000,B 0.000,C 90.000,E1 103.536} C_DIS
LIN {X 0.042,Y -583.982,Z 699.369,A 0.000,B 0.000,C 90.000,E1 102.479} C_DIS
LIN {X -0.133,Y -585.574,Z 699.363,A 0.000,B 0.000,C 90.000,E1 101.422} C_DIS
LIN {X -0.043,Y -587.635,Z 699.356,A 0.000,B 0.000,C 90.000,E1 100.074} C_DIS
LIN {X 0.295,Y -589.145,Z 699.350,A 0.000,B 0.000,C 90.000,E1 98.973} C_DIS
LIN {X 0.249,Y -590.856,Z 699.343,A 0.000,B 0.000,C 90.000,E1 97.644} C_DIS
LIN {X -0.157,Y -592.829,Z 699.334,A 0.000,B 0.000,C 90.000,E1 96.087} C_DIS
LIN {X -0.147,Y -594.402,Z 699.326,A 0.000,B 0.000,C 90.000,E1 94.759} C_DIS
LIN {X -0.212,Y -595.822,Z 699.319,A 0.000,B 0.000,C 90.000,E1 93.440} C_DIS
LIN {X -0.242,Y -597.081,Z 699.312,A 0.000,B 0.000,C 90.000,E1 92.121} C_DIS
LIN {X -0.125,Y -597.782,Z 699.307,A 0.000,B 0.000,C 90.000,E1 91.318} C_DIS
LIN {X -0.143,Y -598.649,Z 699.300,A 0.000,B 0.000,C 90.000,E1 90.000} C_DIS
LIN {X 0.214,Y -599.180,Z 699.294,A 0.000,B 0.000,C 90.000,E1 88.912} C_DIS
LIN {X -0.126,Y -599.667,Z 699.285,A 0.000,B 0.000,C 90.000,E1 87.364} C_DIS
LIN {X -0.100,Y -599.967,Z 699.278,A 0.000,B 0.000,C 90.000,E1 86.045} C_DIS
LIN {X -0.032,Y -600.092,Z 699.271,A 0.000,B 0.000,C 90.000,E1 84.723} C_DIS
LIN {X 0.103,Y -600.041,Z 699.263,A 0.000,B 0.000,C 90.000,E1 83.394} C_DIS
LIN {X -0.051,Y -599.871,Z 699.258,A 0.000,B 0.000,C 90.000,E1 82.356} C_DIS
LIN {X 0.080,Y -599.446,Z 699.250,A 0.000,B 0.000,C 90.000,E1 81.027} C_DIS
LIN {X -0.005,Y -598.858,Z 699.244,A 0.000,B 0.000,C 90.000,E1 79.982} C_DIS
LIN {X 0.301,Y -598.256,Z 699.240,A 0.000,B 0.000,C 90.000,E1 79.162} C_DIS
LIN {X 0.195,Y -597.004,Z 699.231,A 0.000,B 0.000,C 90.000,E1 77.589} C_DIS
LIN {X 0.186,Y -596.013,Z 699.225,A 0.000,B 0.000,C 90.000,E1 76.533} C_DIS
LIN {X -0.286,Y -594.434,Z 699.216,A 0.000,B 0.000,C 90.000,E1 74.991} C_DIS
LIN {X -0.051,Y -592.628,Z 699.208,A 0.000,B 0.000,C 90.000,E1 73.378} C_DIS
LIN {X 0.024,Y -591.297,Z 699.202,A 0.000,B 0.000,C 90.000,E1 72.308} C_DIS
LIN {X 0.255,Y -589.952,Z 699.196,A 0.000,B 0.000,C 90.000,E1 71.221} C_DIS
LIN {X -0.218,Y -587.985,Z 699.188,A 0.000,B 0.000,C 90.000,E1 69.934} C_DIS
LIN {X -0.039,Y -586.276,Z 699.182,A 0.000,B 0.000,C 90.000,E1 68.847} C_DIS
LIN {X 0.124,Y -584.900,Z 699.178,A 0.000,B 0.000,C 90.000,E1 68.028} C_DIS
LIN {X -0.075,Y -582.850,Z 699.172,A 0.000,B 0.000,C 90.000,E1 66.975} C_DIS
LIN {X 0.088,Y -579.907,Z 699.165,A 0.000,B 0.000,C 90.000,E1 65.613} C_DIS
LIN {X 0.193,Y -577.908,Z 699.160,A 0.000,B 0.000,C 90.000,E1 64.793} C_DIS
LIN {X 0.123,Y -574.931,Z 699.154,A 0.000,B 0.000,C 90.000,E1 63.717} C_DIS
LIN {X -0.083,Y -572.522,Z 699.150,A 0.000,B 0.000,C 90.000,E1 62.922} C_DIS
LIN {X 0.038,Y -569.037,Z 699.143,A 0.000,B 0.000,C 90.000,E1 61.820} C_DIS
LIN {X 0.012,Y -566.214,Z 699.139,A 0.000,B 0.000,C 90.000,E1 61.001} C_DIS
LIN {X -0.269,Y -563.135,Z 699.134,A 0.000,B 0.000,C 90.000,E1 60.205} C_DIS
LIN {X 0.190,Y -559.758,Z 699.130,A 0.000,B 0.000,C 90.000,E1 59.331} C_DIS
LIN {X -0.050,Y -556.599,Z 699.126,A 0.000,B 0.000,C 90.000,E1 58.663} C_DIS
LIN {X -0.316,Y -553.086,Z 699.122,A 0.000,B 0.000,C 90.000,E1 57.995} C_DIS
LIN {X 0.022,Y -548.297,Z 699.117,A 0.000,B 0.000,C 90.000,E1 57.120} C_DIS
LIN {X 0.110,Y -544.817,Z 699.114,A 0.000,B 0.000,C 90.000,E1 56.548} C_DIS
LIN {X -0.263,Y -539.945,Z 699.110,A 0.000,B 0.000,C 90.000,E1 55.881} C_DIS
LIN {X -0.081,Y -536.851,Z 699.108,A 0.000,B 0.000,C 90.000,E1 55.435} C_DIS
LIN {X 0.066,Y -532.225,Z 699.105,A 0.000,B 0.000,C 90.000,E1 54.848} C_DIS
LIN {X 0.215,Y -528.367,Z 699.102,A 0.000,B 0.000,C 90.000,E1 54.402} C_DIS
LIN {X -0.008,Y -521.912,Z 699.099,A 0.000,B 0.000,C 90.000,E1 53.783} C_DIS
LIN {X -0.158,Y -517.733,Z 699.097,A 0.000,B 0.000,C 90.000,E1 53.417} C_DIS
LIN {X -0.102,Y -513.158,Z 699.095,A 0.000,B 0.000,C 90.000,E1 53.050} C_DIS
LIN {X 0.207,Y -507.038,Z 699.092,A 0.000,B 0.000,C 90.000,E1 52.557} C_DIS
LIN {X 0.251,Y -500.299,Z 699.090,A 0.000,B 0.000,C 90.000,E1 52.110} C_DIS
LIN {X -0.034,Y -490.535,Z 699.086,A 0.000,B 0.000,C 90.000,E1 51.537} C_DIS
LIN {X -0.001,Y -475.641,Z 699.082,A 0.000,B 0.000,C 90.000,E1 50.678} C_DIS
LIN {X 0.034,Y -459.166,Z 699.076,A 0.000,B 0.000,C 90.000,E1 49.703} C_DIS
LIN {X -0.121,Y -431.799,Z 699.067,A 0.000,B 0.000,C 90.000,E1 48.000} C_DIS
LIN {X -0.146,Y -423.458,Z 699.063,A 0.000,B 0.000,C 90.000,E1 47.391} C_DIS
LIN {X -0.174,Y -423.449,Z 699.063,A 0.000,B 0.000,C 90.000,E1 47.391} C_DIS
LIN {X 0.224,Y -418.864,Z 699.050,A 0.000,B 0.000,C 90.000,E1 44.919} C_DIS
LIN {X -0.003,Y -417.305,Z 699.046,A 0.000,B 0.000,C 90.000,E1 44.271} C_DIS
LIN {X -0.259,Y -410.612,Z 699.029,A 0.000,B 0.000,C 90.000,E1 41.229} C_DIS
LIN {X 0.145,Y -410.790,Z 699.010,A 0.000,B 0.000,C 90.000,E1 37.729} C_DIS
LIN {X -0.046,Y -411.900,Z 698.993,A 0.000,B 0.000,C 90.000,E1 34.659} C_DIS
LIN {X -0.106,Y -412.516,Z 698.985,A 0.000,B 0.000,C 90.000,E1 33.293} C_DIS
LIN {X 0.070,Y -413.571,Z 698.974,A 0.000,B 0.000,C 90.000,E1 31.209} C_DIS
LIN {X 0.065,Y -414.671,Z 698.962,A 0.000,B 0.000,C 90.000,E1 29.155} C_DIS
LIN {X -0.120,Y -415.872,Z 698.951,A 0.000,B 0.000,C 90.000,E1 27.129} C_DIS
LIN {X -0.028,Y -417.774,Z 698.935,A 0.000,B 0.000,C 90.000,E1 24.387} C_DIS
LIN {X -0.072,Y -420.424,Z 698.919,A 0.000,B 0.000,C 90.000,E1 21.334} C_DIS
LIN {X 0.172,Y -422.407,Z 698.907,A 0.000,B 0.000,C 90.000,E1 19.268} C_DIS
LIN {X 0.149,Y -424.173,Z 698.898,A 0.000,B 0.000,C 90.000,E1 17.583} C_DIS
LIN {X 0.160,Y -426.045,Z 698.888,A 0.000,B 0.000,C 90.000,E1 15.898} C_DIS
LIN {X -0.153,Y -428.763,Z 698.875,A 0.000,B 0.000,C 90.000,E1 13.592} C_DIS
LIN {X 0.238,Y -431.256,Z 698.864,A 0.000,B 0.000,C 90.000,E1 11.535} C_DIS
LIN {X 0.096,Y -433.813,Z 698.853,A 0.000,B 0.000,C 90.000,E1 9.557} C_DIS
LIN {X -0.132,Y -437.787,Z 698.837,A 0.000,B 0.000,C 90.000,E1 6.606} C_DIS
LIN {X 0.117,Y -442.025,Z 698.820,A 0.000,B 0.000,C 90.000,E1 3.612} C_DIS
LIN {X -0.153,Y -446.210,Z 698.806,A 0.000,B 0.000,C 90.000,E1 1.031} C_DIS
LIN {X 0.052,Y -451.349,Z 698.790,A 0.000,B 0.000,C 90.000,E1 358.165} C_DIS
LIN {X 0.164,Y -455.030,Z 698.779,A 0.000,B 0.000,C 90.000,E1 356.216} C_DIS
LIN {X -0.039,Y -458.858,Z 698.768,A 0.000,B 0.000,C 90.000,E1 354.318} C_DIS
LIN {X 0.147,Y -460.817,Z 698.763,A 0.000,B 0.000,C 90.000,E1 353.337} C_DIS
LIN {X 0.126,Y -464.557,Z 698.753,A 0.000,B 0.000,C 90.000,E1 351.432} C_DIS
LIN {X 0.253,Y -466.966,Z 698.745,A 0.000,B 0.000,C 90.000,E1 350.151} C_DIS
LIN {X 0.239,Y -469.861,Z 698.737,A 0.000,B 0.000,C 90.000,E1 348.578} C_DIS
LIN {X -0.192,Y -472.710,Z 698.728,A 0.000,B 0.000,C 90.000,E1 347.061} C_DIS
LIN {X -0.067,Y -476.151,Z 698.718,A 0.000,B 0.000,C 90.000,E1 345.172} C_DIS
LIN {X -0.195,Y -479.671,Z 698.707,A 0.000,B 0.000,C 90.000,E1 343.323} C_DIS
LIN {X -0.094,Y -482.707,Z 698.699,A 0.000,B 0.000,C 90.000,E1 341.764} C_DIS
LIN {X 0.228,Y -486.489,Z 698.688,A 0.000,B 0.000,C 90.000,E1 339.880} C_DIS
LIN {X -0.249,Y -490.924,Z 698.677,A 0.000,B 0.000,C 90.000,E1 337.794} C_DIS
LIN {X -0.218,Y -491.543,Z 698.675,A 0.000,B 0.000,C 90.000,E1 337.486} C_DIS
LIN {X 0.044,Y -493.078,Z 698.671,A 0.000,B 0.000,C 90.000,E1 336.847} C_DIS
LIN {X 0.084,Y -493.996,Z 698.670,A 0.000,B 0.000,C 90.000,E1 336.538} C_DIS
LIN {X 0.170,Y -495.195,Z 698.668,A 0.000,B 0.000,C 90.000,E1 336.230} C_DIS
LIN {X 0.215,Y -496.219,Z 698.666,A 0.000,B 0.000,C 90.000,E1 335.921} C_DIS
LIN {X -0.190,Y -497.695,Z 698.665,A 0.000,B 0.000,C 90.000,E1 335.665} C_DIS
LIN {X -0.135,Y -499.760,Z 698.663,A 0.000,B 0.000,C 90.000,E1 335.357} C_DIS
LIN {X 0.122,Y -500.936,Z 698.662,A 0.000,B 0.000,C 90.000,E1 335.177} C_DIS
LIN {X -0.185,Y -503.769,Z 698.661,A 0.000,B 0.000,C 90.000,E1 334.921} C_DIS
LIN {X -0.050,Y -509.231,Z 698.658,A 0.000,B 0.000,C 90.000,E1 334.460} C_DIS
LIN {X 0.039,Y -513.941,Z 698.656,A 0.000,B 0.000,C 90.000,E1 334.101} C_DIS
LIN {X 0.061,Y -531.217,Z 698.650,A 0.000,B 0.000,C 90.000,E1 332.948} C_DIS
LIN {X 0.289,Y -540.263,Z 698.646,A 0.000,B 0.000,C 90.000,E1 332.281} C_DIS
LIN {X 0.080,Y -544.665,Z 698.644,A 0.000,B 0.000,C 90.000,E1 331.975} C_DIS
LIN {X 0.079,Y -550.354,Z 698.642,A 0.000,B 0.000,C 90.000,E1 331.513} C_DIS
LIN {X -0.123,Y -554.540,Z 698.640,A 0.000,B 0.000,C 90.000,E1 331.179} C_DIS
LIN {X 0.125,Y -561.205,Z 698.636,A 0.000,B 0.000,C 90.000,E1 330.539} C_DIS
LIN {X -0.058,Y -568.921,Z 698.632,A 0.000,B 0.000,C 90.000,E1 329.793} C_DIS
LIN {X 0.004,Y -575.242,Z 698.629,A 0.000,B 0.000,C 90.000,E1 329.125} C_DIS
LIN {X -0.133,Y -583.880,Z 698.623,A 0.000,B 0.000,C 90.000,E1 328.201} C_DIS
LIN {X 0.008,Y -589.867,Z 698.620,A 0.000,B 0.000,C 90.000,E1 327.533} C_DIS
LIN {X -0.250,Y -597.980,Z 698.615,A 0.000,B 0.000,C 90.000,E1 326.628} C_DIS
LIN {X 0.174,Y -603.473,Z 698.611,A 0.000,B 0.000,C 90.000,E1 325.928} C_DIS
LIN {X -0.195,Y -608.673,Z 698.607,A 0.000,B 0.000,C 90.000,E1 325.308} C_DIS
LIN {X -0.025,Y -613.597,Z 698.604,A 0.000,B 0.000,C 90.000,E1 324.642} C_DIS
LIN {X 0.067,Y -617.332,Z 698.601,A 0.000,B 0.000,C 90.000,E1 324.116} C_DIS
LIN {X 0.127,Y -623.470,Z 698.596,A 0.000,B 0.000,C 90.000,E1 323.210} C_DIS
LIN {X -0.079,Y -626.835,Z 698.593,A 0.000,B 0.000,C 90.000,E1 322.718} C_DIS
LIN {X -0.046,Y -633.125,Z 698.587,A 0.000,B 0.000,C 90.000,E1 321.698} C_DIS
LIN {X -0.303,Y -636.882,Z 698.584,A 0.000,B 0.000,C 90.000,E1 321.090} C_DIS
LIN {X -0.130,Y -641.931,Z 698.579,A 0.000,B 0.000,C 90.000,E1 320.194} C_DIS
LIN {X 0.101,Y -647.389,Z 698.573,A 0.000,B 0.000,C 90.000,E1 319.175} C_DIS
LIN {X -0.094,Y -651.986,Z 698.568,A 0.000,B 0.000,C 90.000,E1 318.324} C_DIS
LIN {X -0.238,Y -656.328,Z 698.564,A 0.000,B 0.000,C 90.000,E1 317.472} C_DIS
LIN {X 0.142,Y -659.824,Z 698.560,A 0.000,B 0.000,C 90.000,E1 316.701} C_DIS
LIN {X 0.050,Y -665.237,Z 698.553,A 0.000,B 0.000,C 90.000,E1 315.486} C_DIS
LIN {X 0.044,Y -669.080,Z 698.547,A 0.000,B 0.000,C 90.000,E1 314.514} C_DIS
LIN {X 0.118,Y -674.520,Z 698.539,A 0.000,B 0.000,C 90.000,E1 313.056} C_DIS
LIN {X 0.294,Y -678.926,Z 698.533,A 0.000,B 0.000,C 90.000,E1 311.838} C_DIS
LIN {X -0.049,Y -681.386,Z 698.529,A 0.000,B 0.000,C 90.000,E1 311.148} C_DIS
LIN {X 0.195,Y -684.478,Z 698.523,A 0.000,B 0.000,C 90.000,E1 310.172} C_DIS
LIN {X -0.102,Y -686.567,Z 698.519,A 0.000,B 0.000,C 90.000,E1 309.483} C_DIS
LIN {X 0.149,Y -688.498,Z 698.515,A 0.000,B 0.000,C 90.000,E1 308.749} C_DIS
LIN {X -0.175,Y -689.681,Z 698.513,A 0.000,B 0.000,C 90.000,E1 308.302} C_DIS
LIN {X 0.342,Y -692.237,Z 698.506,A 0.000,B 0.000,C 90.000,E1 307.076} C_DIS
LIN {X -0.069,Y -694.474,Z 698.500,A 0.000,B 0.000,C 90.000,E1 305.931} C_DIS
LIN {X -0.157,Y -695.718,Z 698.496,A 0.000,B 0.000,C 90.000,E1 305.231} C_DIS
LIN {X 0.043,Y -697.347,Z 698.489,A 0.000,B 0.000,C 90.000,E1 304.040} C_DIS
LIN {X 0.220,Y -698.489,Z 698.484,A 0.000,B 0.000,C 90.000,E1 303.086} C_DIS
LIN {X 0.414,Y -699.394,Z 698.479,A 0.000,B 0.000,C 90.000,E1 302.133} C_DIS
LIN {X -0.084,Y -700.477,Z 698.472,A 0.000,B 0.000,C 90.000,E1 301.003} C_DIS
LIN {X 0.112,Y -701.009,Z 698.468,A 0.000,B 0.000,C 90.000,E1 300.285} C_DIS
LIN {X 0.258,Y -701.631,Z 698.461,A 0.000,B 0.000,C 90.000,E1 298.871} C_DIS
LIN {X 0.283,Y -702.424,Z 698.450,A 0.000,B 0.000,C 90.000,E1 297.001} C_DIS
LIN {X 0.396,Y -703.194,Z 698.442,A 0.000,B 0.000,C 90.000,E1 295.591} C_DIS
LIN {X 0.022,Y -703.241,Z 698.440,A 0.000,B 0.000,C 90.000,E1 295.155} C_DIS
LIN {X 0.305,Y -702.977,Z 698.439,A 0.000,B 0.000,C 90.000,E1 294.899} C_DIS
LIN {X -0.065,Y -702.032,Z 698.436,A 0.000,B 0.000,C 90.000,E1 294.463} C_DIS
LIN {X 0.213,Y -700.890,Z 698.435,A 0.000,B 0.000,C 90.000,E1 294.207} C_DIS
LIN {X -0.152,Y -699.293,Z 698.433,A 0.000,B 0.000,C 90.000,E1 294.003} C_DIS
LIN {X -0.168,Y -697.442,Z 698.432,A 0.000,B 0.000,C 90.000,E1 293.770} C_DIS
LIN {X -0.037,Y -696.246,Z 698.431,A 0.000,B 0.000,C 90.000,E1 293.643} C_DIS
LIN {X 0.094,Y -694.383,Z 698.431,A 0.000,B 0.000,C 90.000,E1 293.515} C_DIS
LIN {X 0.054,Y -688.706,Z 698.429,A 0.000,B 0.000,C 90.000,E1 293.259} C_DIS
LIN {X -0.207,Y -686.632,Z 698.429,A 0.000,B 0.000,C 90.000,E1 293.206} C_DIS
LIN {X -0.036,Y -684.443,Z 698.429,A 0.000,B 0.000,C 90.000,E1 293.131} C_DIS
LIN {X -0.172,Y -677.780,Z 698.428,A 0.000,B 0.000,C 90.000,E1 293.003} C_DIS
LIN {X 0.175,Y -661.374,Z 698.427,A 0.000,B 0.000,C 90.000,E1 292.770} C_DIS
LIN {X -0.184,Y -647.634,Z 698.425,A 0.000,B 0.000,C 90.000,E1 292.589} C_DIS
LIN {X 0.019,Y -637.805,Z 698.424,A 0.000,B 0.000,C 90.000,E1 292.386} C_DIS
LIN {X 0.103,Y -624.561,Z 698.423,A 0.000,B 0.000,C 90.000,E1 292.078} C_DIS
LIN {X -0.111,Y -607.450,Z 698.420,A 0.000,B 0.000,C 90.000,E1 291.642} C_DIS
LIN {X 0.078,Y -576.520,Z 698.415,A 0.000,B 0.000,C 90.000,E1 290.684} C_DIS
LIN {X 0.013,Y -568.905,Z 698.414,A 0.000,B 0.000,C 90.000,E1 290.482} C_DIS
LIN {X -0.157,Y -561.736,Z 698.412,A 0.000,B 0.000,C 90.000,E1 290.248} C_DIS
LIN {X 0.229,Y -558.688,Z 698.412,A 0.000,B 0.000,C 90.000,E1 290.066} C_DIS
LIN {X -0.125,Y -555.781,Z 698.410,A 0.000,B 0.000,C 90.000,E1 289.866} C_DIS
LIN {X -0.154,Y -555.767,Z 698.410,A 0.000,B 0.000,C 90.000,E1 289.866} C_DIS
LIN {X -0.022,Y -554.945,Z 698.409,A 0.000,B 0.000,C 90.000,E1 289.631} C_DIS
LIN {X -0.275,Y -554.496,Z 698.407,A 0.000,B 0.000,C 90.000,E1 289.268} C_DIS
LIN {X -0.166,Y -553.869,Z 698.398,A 0.000,B 0.000,C 90.000,E1 287.583} C_DIS
LIN {X -0.076,Y -553.235,Z 698.388,A 0.000,B 0.000,C 90.000,E1 285.898} C_DIS
LIN {X 0.115,Y -552.738,Z 698.381,A 0.000,B 0.000,C 90.000,E1 284.481} C_DIS
LIN {X -0.235,Y -552.229,Z 698.373,A 0.000,B 0.000,C 90.000,E1 283.119} C_DIS
LIN {X -0.183,Y -551.610,Z 698.365,A 0.000,B 0.000,C 90.000,E1 281.715} C_DIS
LIN {X -0.143,Y -550.969,Z 698.357,A 0.000,B 0.000,C 90.000,E1 280.310} C_DIS
LIN {X 0.028,Y -550.051,Z 698.345,A 0.000,B 0.000,C 90.000,E1 278.049} C_DIS
LIN {X 0.138,Y -549.276,Z 698.331,A 0.000,B 0.000,C 90.000,E1 275.511} C_DIS
LIN {X 0.038,Y -549.004,Z 698.320,A 0.000,B 0.000,C 90.000,E1 273.555} C_DIS
LIN {X 0.262,Y -548.798,Z 698.314,A 0.000,B 0.000,C 90.000,E1 272.407} C_DIS
LIN {X -0.019,Y -548.328,Z 698.306,A 0.000,B 0.000,C 90.000,E1 271.031} C_DIS
LIN {X -0.274,Y -547.425,Z 698.296,A 0.000,B 0.000,C 90.000,E1 269.370} C_DIS
LIN {X 0.051,Y -546.232,Z 698.285,A 0.000,B 0.000,C 90.000,E1 267.364} C_DIS
LIN {X -0.208,Y -545.117,Z 698.276,A 0.000,B 0.000,C 90.000,E1 265.698} C_DIS
LIN {X 0.197,Y -543.430,Z 698.263,A 0.000,B 0.000,C 90.000,E1 263.394} C_DIS
LIN {X -0.085,Y -542.099,Z 698.256,A 0.000,B 0.000,C 90.000,E1 262.008} C_DIS
LIN {X 0.207,Y -540.426,Z 698.246,A 0.000,B 0.000,C 90.000,E1 260.274} C_DIS
LIN {X 0.113,Y -538.860,Z 698.237,A 0.000,B 0.000,C 90.000,E1 258.578} C_DIS
LIN {X -0.075,Y -537.587,Z 698.229,A 0.000,B 0.000,C 90.000,E1 257.173} C_DIS
LIN {X -0.053,Y -535.869,Z 698.218,A 0.000,B 0.000,C 90.000,E1 255.172} C_DIS
LIN {X 0.003,Y -534.130,Z 698.208,A 0.000,B 0.000,C 90.000,E1 253.449} C_DIS
LIN {X -0.144,Y -532.051,Z 698.197,A 0.000,B 0.000,C 90.000,E1 251.456} C_DIS
LIN {X -0.049,Y -530.874,Z 698.191,A 0.000,B 0.000,C 90.000,E1 250.296} C_DIS
LIN {X -0.158,Y -529.847,Z 698.186,A 0.000,B 0.000,C 90.000,E1 249.444} C_DIS
LIN {X 0.085,Y -527.854,Z 698.178,A 0.000,B 0.000,C 90.000,E1 247.975} C_DIS
LIN {X -0.001,Y -525.771,Z 698.170,A 0.000,B 0.000,C 90.000,E1 246.538} C_DIS
LIN {X 0.190,Y -523.909,Z 698.163,A 0.000,B 0.000,C 90.000,E1 245.357} C_DIS
LIN {X 0.246,Y -521.482,Z 698.155,A 0.000,B 0.000,C 90.000,E1 243.896} C_DIS
LIN {X -0.211,Y -518.686,Z 698.147,A 0.000,B 0.000,C 90.000,E1 242.487} C_DIS
LIN {X -0.023,Y -515.825,Z 698.139,A 0.000,B 0.000,C 90.000,E1 241.001} C_DIS
LIN {X 0.260,Y -513.419,Z 698.132,A 0.000,B 0.000,C 90.000,E1 239.793} C_DIS
LIN {X -0.210,Y -509.655,Z 698.123,A 0.000,B 0.000,C 90.000,E1 238.074} C_DIS
LIN {X -0.123,Y -506.423,Z 698.114,A 0.000,B 0.000,C 90.000,E1 236.580} C_DIS
LIN {X -0.234,Y -503.122,Z 698.106,A 0.000,B 0.000,C 90.000,E1 235.102} C_DIS
LIN {X 0.127,Y -500.382,Z 698.099,A 0.000,B 0.000,C 90.000,E1 233.863} C_DIS
LIN {X 0.059,Y -498.203,Z 698.094,A 0.000,B 0.000,C 90.000,E1 232.970} C_DIS
LIN {X -0.042,Y -493.576,Z 698.084,A 0.000,B 0.000,C 90.000,E1 231.170} C_DIS
LIN {X 0.048,Y -489.155,Z 698.074,A 0.000,B 0.000,C 90.000,E1 229.337} C_DIS
LIN {X -0.240,Y -484.186,Z 698.062,A 0.000,B 0.000,C 90.000,E1 227.229} C_DIS
LIN {X 0.028,Y -479.367,Z 698.050,A 0.000,B 0.000,C 90.000,E1 225.040} C_DIS
LIN {X 0.166,Y -476.579,Z 698.043,A 0.000,B 0.000,C 90.000,E1 223.785} C_DIS
LIN {X 0.229,Y -471.735,Z 698.031,A 0.000,B 0.000,C 90.000,E1 221.595} C_DIS
LIN {X -0.098,Y -466.926,Z 698.019,A 0.000,B 0.000,C 90.000,E1 219.439} C_DIS
LIN {X 0.141,Y -464.978,Z 698.014,A 0.000,B 0.000,C 90.000,E1 218.463} C_DIS
LIN {X -0.033,Y -460.940,Z 698.003,A 0.000,B 0.000,C 90.000,E1 216.583} C_DIS
LIN {X -0.099,Y -455.995,Z 697.989,A 0.000,B 0.000,C 90.000,E1 214.040} C_DIS
LIN {X 0.127,Y -452.322,Z 697.978,A 0.000,B 0.000,C 90.000,E1 212.084} C_DIS
LIN {X -0.265,Y -448.045,Z 697.966,A 0.000,B 0.000,C 90.000,E1 209.873} C_DIS
LIN {X -0.066,Y -444.487,Z 697.955,A 0.000,B 0.000,C 90.000,E1 207.897} C_DIS
LIN {X 0.183,Y -441.528,Z 697.946,A 0.000,B 0.000,C 90.000,E1 206.232} C_DIS
LIN {X 0.204,Y -437.992,Z 697.935,A 0.000,B 0.000,C 90.000,E1 204.259} C_DIS
LIN {X -0.215,Y -434.326,Z 697.924,A 0.000,B 0.000,C 90.000,E1 202.333} C_DIS
LIN {X 0.049,Y -431.931,Z 697.917,A 0.000,B 0.000,C 90.000,E1 200.972} C_DIS
LIN {X -0.062,Y -427.679,Z 697.904,A 0.000,B 0.000,C 90.000,E1 198.652} C_DIS
LIN {X -0.088,Y -422.838,Z 697.889,A 0.000,B 0.000,C 90.000,E1 195.969} C_DIS
LIN {X 0.164,Y -419.805,Z 697.879,A 0.000,B 0.000,C 90.000,E1 194.245} C_DIS
LIN {X -0.104,Y -416.246,Z 697.868,A 0.000,B 0.000,C 90.000,E1 192.243} C_DIS
LIN {X -0.137,Y -412.809,Z 697.857,A 0.000,B 0.000,C 90.000,E1 190.197} C_DIS
LIN {X 0.078,Y -409.468,Z 697.845,A 0.000,B 0.000,C 90.000,E1 188.106} C_DIS
LIN {X 0.100,Y -406.389,Z 697.834,A 0.000,B 0.000,C 90.000,E1 186.030} C_DIS
LIN {X 0.042,Y -403.446,Z 697.822,A 0.000,B 0.000,C 90.000,E1 183.955} C_DIS
LIN {X 0.063,Y -399.116,Z 697.803,A 0.000,B 0.000,C 90.000,E1 180.458} C_DIS
LIN {X -0.131,Y -395.399,Z 697.781,A 0.000,B 0.000,C 90.000,E1 176.617} C_DIS
LIN {X -0.159,Y -393.616,Z 697.767,A 0.000,B 0.000,C 90.000,E1 174.147} C_DIS
LIN {X 0.086,Y -392.048,Z 697.748,A 0.000,B 0.000,C 90.000,E1 170.566} C_DIS
LIN {X -0.143,Y -391.244,Z 697.732,A 0.000,B 0.000,C 90.000,E1 167.757} C_DIS
LIN {X 0.151,Y -390.782,Z 697.722,A 0.000,B 0.000,C 90.000,E1 165.936} C_DIS
LIN {X 0.159,Y -390.281,Z 697.706,A 0.000,B 0.000,C 90.000,E1 163.087} C_DIS
LIN {X 0.043,Y -390.209,Z 697.694,A 0.000,B 0.000,C 90.000,E1 160.967} C_DIS
LIN {X 0.103,Y -390.252,Z 697.680,A 0.000,B 0.000,C 90.000,E1 158.465} C_DIS
LIN {X -0.101,Y -390.405,Z 697.669,A 0.000,B 0.000,C 90.000,E1 156.357} C_DIS
LIN {X 0.039,Y -390.728,Z 697.655,A 0.000,B 0.000,C 90.000,E1 153.845} C_DIS
LIN {X -0.024,Y -390.997,Z 697.643,A 0.000,B 0.000,C 90.000,E1 151.719} C_DIS
LIN {X 0.047,Y -392.002,Z 697.623,A 0.000,B 0.000,C 90.000,E1 148.152} C_DIS
LIN {X 0.016,Y -393.824,Z 697.603,A 0.000,B 0.000,C 90.000,E1 144.609} C_DIS
LIN {X 0.043,Y -394.473,Z 697.598,A 0.000,B 0.000,C 90.000,E1 143.543} C_DIS
LIN {X 0.023,Y -395.982,Z 697.588,A 0.000,B 0.000,C 90.000,E1 141.778} C_DIS
LIN {X 0.109,Y -398.365,Z 697.574,A 0.000,B 0.000,C 90.000,E1 139.299} C_DIS
LIN {X 0.044,Y -400.302,Z 697.564,A 0.000,B 0.000,C 90.000,E1 137.553} C_DIS
LIN {X -0.034,Y -401.060,Z 697.560,A 0.000,B 0.000,C 90.000,E1 136.863} C_DIS
LIN {X -0.008,Y -402.880,Z 697.555,A 0.000,B 0.000,C 90.000,E1 135.810} C_DIS
LIN {X -0.160,Y -404.990,Z 697.550,A 0.000,B 0.000,C 90.000,E1 135.081} C_DIS
LIN {X -0.043,Y -406.554,Z 697.548,A 0.000,B 0.000,C 90.000,E1 134.717} C_DIS
LIN {X 0.163,Y -407.234,Z 697.547,A 0.000,B 0.000,C 90.000,E1 134.514} C_DIS
LIN {X 0.003,Y -409.464,Z 697.546,A 0.000,B 0.000,C 90.000,E1 134.190} C_DIS
LIN {X -0.153,Y -412.263,Z 697.544,A 0.000,B 0.000,C 90.000,E1 133.866} C_DIS
LIN {X -0.162,Y -415.209,Z 697.542,A 0.000,B 0.000,C 90.000,E1 133.542} C_DIS
LIN {X -0.087,Y -420.842,Z 697.539,A 0.000,B 0.000,C 90.000,E1 132.975} C_DIS
LIN {X -0.203,Y -436.144,Z 697.531,A 0.000,B 0.000,C 90.000,E1 131.595} C_DIS
LIN {X 0.131,Y -449.954,Z 697.524,A 0.000,B 0.000,C 90.000,E1 130.378} C_DIS
LIN {X -0.058,Y -457.630,Z 697.521,A 0.000,B 0.000,C 90.000,E1 129.769} C_DIS
LIN {X 0.059,Y -465.283,Z 697.517,A 0.000,B 0.000,C 90.000,E1 129.116} C_DIS
LIN {X -0.092,Y -475.600,Z 697.512,A 0.000,B 0.000,C 90.000,E1 128.222} C_DIS
LIN {X -0.047,Y -481.336,Z 697.509,A 0.000,B 0.000,C 90.000,E1 127.684} C_DIS
LIN {X -0.093,Y -489.906,Z 697.505,A 0.000,B 0.000,C 90.000,E1 126.870} C_DIS
LIN {X -0.008,Y -496.761,Z 697.501,A 0.000,B 0.000,C 90.000,E1 126.171} C_DIS
LIN {X 0.067,Y -502.149,Z 697.498,A 0.000,B 0.000,C 90.000,E1 125.598} C_DIS
LIN {X -0.067,Y -506.035,Z 697.495,A 0.000,B 0.000,C 90.000,E1 125.185} C_DIS
LIN {X -0.035,Y -510.989,Z 697.492,A 0.000,B 0.000,C 90.000,E1 124.612} C_DIS
LIN {X -0.314,Y -514.697,Z 697.490,A 0.000,B 0.000,C 90.000,E1 124.199} C_DIS
LIN {X 0.141,Y -518.245,Z 697.487,A 0.000,B 0.000,C 90.000,E1 123.706} C_DIS
LIN {X -0.274,Y -522.554,Z 697.484,A 0.000,B 0.000,C 90.000,E1 123.166} C_DIS
LIN {X 0.065,Y -526.556,Z 697.481,A 0.000,B 0.000,C 90.000,E1 122.546} C_DIS
LIN {X -0.294,Y -530.358,Z 697.478,A 0.000,B 0.000,C 90.000,E1 122.005} C_DIS
LIN {X -0.044,Y -534.538,Z 697.474,A 0.000,B 0.000,C 90.000,E1 121.258} C_DIS
LIN {X -0.082,Y -538.969,Z 697.469,A 0.000,B 0.000,C 90.000,E1 120.413} C_DIS
LIN {X -0.360,Y -541.740,Z 697.466,A 0.000,B 0.000,C 90.000,E1 119.873} C_DIS
LIN {X -0.140,Y -545.596,Z 697.461,A 0.000,B 0.000,C 90.000,E1 118.999} C_DIS
LIN {X -0.025,Y -548.649,Z 697.457,A 0.000,B 0.000,C 90.000,E1 118.281} C_DIS
LIN {X -0.002,Y -552.044,Z 697.452,A 0.000,B 0.000,C 90.000,E1 117.436} C_DIS
LIN {X -0.197,Y -555.212,Z 697.448,A 0.000,B 0.000,C 90.000,E1 116.616} C_DIS
LIN {X 0.181,Y -559.128,Z 697.442,A 0.000,B 0.000,C 90.000,E1 115.463} C_DIS
LIN {X 0.068,Y -561.777,Z 697.437,A 0.000,B 0.000,C 90.000,E1 114.643} C_DIS
LIN {X -0.017,Y -564.174,Z 697.432,A 0.000,B 0.000,C 90.000,E1 113.823} C_DIS
LIN {X -0.083,Y -566.242,Z 697.428,A 0.000,B 0.000,C 90.000,E1 113.003} C_DIS
LIN {X -0.160,Y -567.577,Z 697.425,A 0.000,B 0.000,C 90.000,E1 112.461} C_DIS
LIN {X -0.059,Y -569.722,Z 697.419,A 0.000,B 0.000,C 90.000,E1 111.354} C_DIS
LIN {X -0.108,Y -572.237,Z 697.411,A 0.000,B 0.000,C 90.000,E1 109.993} C_DIS
LIN {X -0.140,Y -574.141,Z 697.405,A 0.000,B 0.000,C 90.000,E1 108.906} C_DIS
LIN {X -0.135,Y -576.899,Z 697.396,A 0.000,B 0.000,C 90.000,E1 107.275} C_DIS
LIN {X 0.099,Y -579.152,Z 697.388,A 0.000,B 0.000,C 90.000,E1 105.898} C_DIS
LIN {X -0.122,Y -581.635,Z 697.379,A 0.000,B 0.000,C 90.000,E1 104.300} C_DIS
LIN {X 0.272,Y -584.117,Z 697.370,A 0.000,B 0.000,C 90.000,E1 102.647} C_DIS
LIN {X 0.340,Y -586.125,Z 697.363,A 0.000,B 0.000,C 90.000,E1 101.299} C_DIS
LIN {X -0.249,Y -588.205,Z 697.356,A 0.000,B 0.000,C 90.000,E1 100.018} C_DIS
LIN {X 0.099,Y -589.724,Z 697.350,A 0.000,B 0.000,C 90.000,E1 98.916} C_DIS
LIN {X 0.064,Y -591.463,Z 697.342,A 0.000,B 0.000,C 90.000,E1 97.587} C_DIS
LIN {X -0.265,Y -593.481,Z 697.333,A 0.000,B 0.000,C 90.000,E1 96.024} C_DIS
LIN {X 0.287,Y -595.037,Z 697.326,A 0.000,B 0.000,C 90.000,E1 94.645} C_DIS
LIN {X 0.237,Y -596.487,Z 697.319,A 0.000,B 0.000,C 90.000,E1 93.326} C_DIS
LIN {X 0.221,Y -597.753,Z 697.311,A 0.000,B 0.000,C 90.000,E1 92.007} C_DIS
LIN {X -0.018,Y -598.594,Z 697.305,A 0.000,B 0.000,C 90.000,E1 90.974} C_DIS
LIN {X -0.261,Y -599.281,Z 697.300,A 0.000,B 0.000,C 90.000,E1 89.943} C_DIS
LIN {X 0.106,Y -599.798,Z 697.294,A 0.000,B 0.000,C 90.000,E1 88.854} C_DIS
LIN {X -0.222,Y -600.302,Z 697.285,A 0.000,B 0.000,C 90.000,E1 87.306} C_DIS
LIN {X -0.187,Y -600.572,Z 697.278,A 0.000,B 0.000,C 90.000,E1 85.988} C_DIS
LIN {X -0.109,Y -600.663,Z 697.270,A 0.000,B 0.000,C 90.000,E1 84.666} C_DIS
LIN {X 0.035,Y -600.591,Z 697.263,A 0.000,B 0.000,C 90.000,E1 83.337} C_DIS
LIN {X -0.114,Y -600.406,Z 697.257,A 0.000,B 0.000,C 90.000,E1 82.299} C_DIS
LIN {X -0.184,Y -600.094,Z 697.251,A 0.000,B 0.000,C 90.000,E1 81.254} C_DIS
LIN {X -0.253,Y -599.507,Z 697.246,A 0.000,B 0.000,C 90.000,E1 80.208} C_DIS
LIN {X 0.255,Y -598.705,Z 697.240,A 0.000,B 0.000,C 90.000,E1 79.106} C_DIS
LIN {X 0.282,Y -597.394,Z 697.231,A 0.000,B 0.000,C 90.000,E1 77.521} C_DIS
LIN {X -0.002,Y -596.666,Z 697.227,A 0.000,B 0.000,C 90.000,E1 76.756} C_DIS
LIN {X -0.166,Y -594.747,Z 697.216,A 0.000,B 0.000,C 90.000,E1 74.921} C_DIS
LIN {X -0.084,Y -592.909,Z 697.207,A 0.000,B 0.000,C 90.000,E1 73.323} C_DIS
LIN {X 0.172,Y -591.589,Z 697.201,A 0.000,B 0.000,C 90.000,E1 72.236} C_DIS
LIN {X 0.096,Y -589.741,Z 697.194,A 0.000,B 0.000,C 90.000,E1 70.913} C_DIS
LIN {X -0.156,Y -587.340,Z 697.185,A 0.000,B 0.000,C 90.000,E1 69.337} C_DIS
LIN {X 0.216,Y -585.470,Z 697.179,A 0.000,B 0.000,C 90.000,E1 68.230} C_DIS
LIN {X 0.018,Y -583.432,Z 697.173,A 0.000,B 0.000,C 90.000,E1 67.177} C_DIS
LIN {X 0.025,Y -581.006,Z 697.167,A 0.000,B 0.000,C 90.000,E1 66.102} C_DIS
LIN {X 0.146,Y -579.106,Z 697.163,A 0.000,B 0.000,C 90.000,E1 65.281} C_DIS
LIN {X 0.247,Y -577.000,Z 697.158,A 0.000,B 0.000,C 90.000,E1 64.460} C_DIS
LIN {X 0.322,Y -574.708,Z 697.154,A 0.000,B 0.000,C 90.000,E1 63.640} C_DIS
LIN {X -0.144,Y -572.237,Z 697.149,A 0.000,B 0.000,C 90.000,E1 62.871} C_DIS
LIN {X -0.032,Y -568.683,Z 697.143,A 0.000,B 0.000,C 90.000,E1 61.769} C_DIS
LIN {X 0.209,Y -565.782,Z 697.139,A 0.000,B 0.000,C 90.000,E1 60.923} C_DIS
LIN {X -0.074,Y -562.623,Z 697.134,A 0.000,B 0.000,C 90.000,E1 60.127} C_DIS
LIN {X 0.095,Y -559.094,Z 697.129,A 0.000,B 0.000,C 90.000,E1 59.282} C_DIS
LIN {X -0.152,Y -555.824,Z 697.126,A 0.000,B 0.000,C 90.000,E1 58.614} C_DIS
LIN {X -0.018,Y -552.979,Z 697.122,A 0.000,B 0.000,C 90.000,E1 58.043} C_DIS
LIN {X 0.148,Y -548.972,Z 697.119,A 0.000,B 0.000,C 90.000,E1 57.327} C_DIS
LIN {X 0.130,Y -544.586,Z 697.115,A 0.000,B 0.000,C 90.000,E1 56.628} C_DIS
LIN {X -0.107,Y -540.700,Z 697.112,A 0.000,B 0.000,C 90.000,E1 56.087} C_DIS
LIN {X -0.039,Y -536.806,Z 697.109,A 0.000,B 0.000,C 90.000,E1 55.548} C_DIS
LIN {X -0.028,Y -532.113,Z 697.105,A 0.000,B 0.000,C 90.000,E1 54.975} C_DIS
LIN {X 0.054,Y -526.851,Z 697.102,A 0.000,B 0.000,C 90.000,E1 54.402} C_DIS
LIN {X 0.088,Y -522.746,Z 697.100,A 0.000,B 0.000,C 90.000,E1 53.989} C_DIS
LIN {X -0.232,Y -516.809,Z 697.097,A 0.000,B 0.000,C 90.000,E1 53.497} C_DIS
LIN {X -0.114,Y -510.458,Z 697.094,A 0.000,B 0.000,C 90.000,E1 53.004} C_DIS
LIN {X 0.130,Y -505.750,Z 697.093,A 0.000,B 0.000,C 90.000,E1 52.637} C_DIS
LIN {X 0.309,Y -499.112,Z 697.090,A 0.000,B 0.000,C 90.000,E1 52.190} C_DIS
LIN {X 0.071,Y -489.285,Z 697.087,A 0.000,B 0.000,C 90.000,E1 51.618} C_DIS
LIN {X 0.074,Y -477.581,Z 697.083,A 0.000,B 0.000,C 90.000,E1 50.964} C_DIS
LIN {X 0.036,Y -471.489,Z 697.081,A 0.000,B 0.000,C 90.000,E1 50.598} C_DIS
LIN {X -0.110,Y -456.650,Z 697.076,A 0.000,B 0.000,C 90.000,E1 49.747} C_DIS
LIN {X -0.026,Y -435.294,Z 697.069,A 0.000,B 0.000,C 90.000,E1 48.405} C_DIS
LIN {X 0.246,Y -432.090,Z 697.068,A 0.000,B 0.000,C 90.000,E1 48.162} C_DIS
LIN {X -0.069,Y -423.943,Z 697.064,A 0.000,B 0.000,C 90.000,E1 47.595} C_DIS
LIN {X 0.217,Y -423.898,Z 697.064,A 0.000,B 0.000,C 90.000,E1 47.553} C_DIS
LIN {X 0.047,Y -418.683,Z 697.049,A 0.000,B 0.000,C 90.000,E1 44.838} C_DIS
LIN {X -0.027,Y -411.077,Z 697.030,A 0.000,B 0.000,C 90.000,E1 41.434} C_DIS
LIN {X 0.136,Y -410.925,Z 697.028,A 0.000,B 0.000,C 90.000,E1 41.067} C_DIS
LIN {X -0.194,Y -411.177,Z 697.011,A 0.000,B 0.000,C 90.000,E1 38.016} C_DIS
LIN {X 0.130,Y -412.395,Z 696.992,A 0.000,B 0.000,C 90.000,E1 34.532} C_DIS
LIN {X 0.082,Y -413.023,Z 696.984,A 0.000,B 0.000,C 90.000,E1 33.166} C_DIS
LIN {X -0.080,Y -414.082,Z 696.973,A 0.000,B 0.000,C 90.000,E1 31.131} C_DIS
LIN {X -0.079,Y -415.214,Z 696.962,A 0.000,B 0.000,C 90.000,E1 29.077} C_DIS
LIN {X 0.055,Y -416.654,Z 696.948,A 0.000,B 0.000,C 90.000,E1 26.668} C_DIS
LIN {X -0.010,Y -418.604,Z 696.933,A 0.000,B 0.000,C 90.000,E1 23.951} C_DIS
LIN {X 0.048,Y -421.012,Z 696.918,A 0.000,B 0.000,C 90.000,E1 21.227} C_DIS
LIN {X 0.135,Y -422.676,Z 696.909,A 0.000,B 0.000,C 90.000,E1 19.523} C_DIS
LIN {X -0.150,Y -424.376,Z 696.899,A 0.000,B 0.000,C 90.000,E1 17.873} C_DIS
LIN {X -0.067,Y -426.545,Z 696.888,A 0.000,B 0.000,C 90.000,E1 15.843} C_DIS
LIN {X -0.044,Y -428.848,Z 696.877,A 0.000,B 0.000,C 90.000,E1 13.828} C_DIS
LIN {X -0.071,Y -431.326,Z 696.866,A 0.000,B 0.000,C 90.000,E1 11.827} C_DIS
LIN {X -0.213,Y -433.820,Z 696.855,A 0.000,B 0.000,C 90.000,E1 9.849} C_DIS
LIN {X 0.048,Y -437.744,Z 696.838,A 0.000,B 0.000,C 90.000,E1 6.834} C_DIS
LIN {X 0.032,Y -440.943,Z 696.825,A 0.000,B 0.000,C 90.000,E1 4.531} C_DIS
LIN {X 0.013,Y -446.080,Z 696.807,A 0.000,B 0.000,C 90.000,E1 1.260} C_DIS
LIN {X 0.056,Y -451.557,Z 696.790,A 0.000,B 0.000,C 90.000,E1 358.165} C_DIS
LIN {X 0.172,Y -455.217,Z 696.779,A 0.000,B 0.000,C 90.000,E1 356.216} C_DIS
LIN {X 0.154,Y -459.686,Z 696.767,A 0.000,B 0.000,C 90.000,E1 353.976} C_DIS
LIN {X 0.128,Y -462.213,Z 696.760,A 0.000,B 0.000,C 90.000,E1 352.704} C_DIS
LIN {X -0.057,Y -465.307,Z 696.751,A 0.000,B 0.000,C 90.000,E1 351.141} C_DIS
LIN {X 0.083,Y -467.683,Z 696.744,A 0.000,B 0.000,C 90.000,E1 349.859} C_DIS
LIN {X -0.098,Y -471.112,Z 696.733,A 0.000,B 0.000,C 90.000,E1 347.993} C_DIS
LIN {X 0.058,Y -473.932,Z 696.725,A 0.000,B 0.000,C 90.000,E1 346.408} C_DIS
LIN {X -0.080,Y -476.852,Z 696.716,A 0.000,B 0.000,C 90.000,E1 344.866} C_DIS
LIN {X 0.118,Y -481.027,Z 696.704,A 0.000,B 0.000,C 90.000,E1 342.670} C_DIS
LIN {X -0.213,Y -485.320,Z 696.692,A 0.000,B 0.000,C 90.000,E1 340.550} C_DIS
LIN {X -0.291,Y -489.072,Z 696.682,A 0.000,B 0.000,C 90.000,E1 338.720} C_DIS
LIN {X -0.123,Y -493.403,Z 696.671,A 0.000,B 0.000,C 90.000,E1 336.719} C_DIS
LIN {X 0.125,Y -493.833,Z 696.670,A 0.000,B 0.000,C 90.000,E1 336.538} C_DIS
LIN {X -0.048,Y -494.618,Z 696.669,A 0.000,B 0.000,C 90.000,E1 336.357} C_DIS
LIN {X 0.043,Y -496.481,Z 696.665,A 0.000,B 0.000,C 90.000,E1 335.741} C_DIS
LIN {X 0.092,Y -497.918,Z 696.664,A 0.000,B 0.000,C 90.000,E1 335.433} C_DIS
LIN {X 0.101,Y -498.703,Z 696.663,A 0.000,B 0.000,C 90.000,E1 335.281} C_DIS
LIN {X 0.159,Y -500.797,Z 696.661,A 0.000,B 0.000,C 90.000,E1 334.973} C_DIS
LIN {X -0.045,Y -505.333,Z 696.659,A 0.000,B 0.000,C 90.000,E1 334.537} C_DIS
